LIN {X 0,Y 350.473,Z 637.276,A -85,B 0,C 180,E1 -13786.754,E2 -13786.754} C_VEL
LIN {X 0,Y 351.298,Z 630.032,A -85,B 0,C 180,E1 -13787.613,E2 -13787.613} C_VEL
LIN {X 0,Y 351.494,Z 617.509,A -85,B 0,C 180,E1 -13788.907,E2 -13788.907} C_VEL
LIN {X 0,Y 351.425,Z 604.758,A -85,B 0,C 180,E1 -13789.96,E2 -13789.96} C_VEL
LIN {X 0,Y 350.462,Z 591.602,A -85,B 0,C 180,E1 -13790.852,E2 -13790.852} C_VEL
LIN {X 0,Y 348.459,Z 578.111,A -85,B 0,C 180,E1 -13791.619,E2 -13791.619} C_VEL
LIN {X 0,Y 347.444,Z 572.402,A -85,B 0,C 180,E1 -13791.906,E2 -13791.906} C_VEL
LIN {X 0,Y 348.181,Z 560.578,A -85,B 0,C 180,E1 -13795.72,E2 -13795.72} C_VEL
LIN {X 0,Y 349.049,Z 549.243,A -85,B 0,C 180,E1 -13799.49,E2 -13799.49} C_VEL
LIN {X 0,Y 350.264,Z 537.694,A -85,B 0,C 180,E1 -13803.49,E2 -13803.49} C_VEL
LIN {X 0,Y 351.508,Z 528.335,A -85,B 0,C 180,E1 -13806.893,E2 -13806.893} C_VEL
LIN {X 0,Y 351.566,Z 524.747,A -85,B 0,C 180,E1 -13808.295,E2 -13808.295} C_VEL
LIN {X 0,Y 350.338,Z 517.421,A -85,B 0,C 180,E1 -13811.453,E2 -13811.453} C_VEL
LIN {X 0,Y 348.766,Z 509.758,A -85,B 0,C 180,E1 -13815.147,E2 -13815.147} C_VEL
LIN {X 0,Y 347.773,Z 505.172,A -85,B 0,C 180,E1 -13817.686,E2 -13817.686} C_VEL
LIN {X 0,Y 347.754,Z 505.168,A -85,B 0,C 180,E1 -13821.208,E2 -13821.208} C_VEL
LIN {X 0,Y 347.79,Z 505.161,A -85,B 0,C 180,E1 -13824.125,E2 -13824.125} C_VEL
LIN {X 0,Y 347.741,Z 505.165,A -85,B 0,C 180,E1 -13828.086,E2 -13828.086} C_VEL
LIN {X 0,Y 347.807,Z 505.155,A -85,B 0,C 180,E1 -13830.99,E2 -13830.99} C_VEL
LIN {X 0,Y 347.834,Z 505.151,A -85,B 0,C 180,E1 -13833.608,E2 -13833.608} C_VEL
LIN {X 0,Y 347.791,Z 505.156,A -85,B 0,C 180,E1 -13836.162,E2 -13836.162} C_VEL
LIN {X 0,Y 347.816,Z 505.157,A -85,B 0,C 180,E1 -13839.91,E2 -13839.91} C_VEL
LIN {X 0,Y 347.869,Z 505.148,A -85,B 0,C 180,E1 -13842.36,E2 -13842.36} C_VEL
LIN {X 0,Y 347.901,Z 505.146,A -85,B 0,C 180,E1 -13845.971,E2 -13845.971} C_VEL
LIN {X 0,Y 347.932,Z 505.144,A -85,B 0,C 180,E1 -13849.526,E2 -13849.526} C_VEL
LIN {X 0,Y 348.078,Z 505.121,A -85,B 0,C 180,E1 -13851.875,E2 -13851.875} C_VEL
LIN {X 0,Y 348.07,Z 505.128,A -85,B 0,C 180,E1 -13854.206,E2 -13854.206} C_VEL
LIN {X 0,Y 348.199,Z 505.111,A -85,B 0,C 180,E1 -13857.687,E2 -13857.687} C_VEL
LIN {X 0,Y 348.327,Z 505.096,A -85,B 0,C 180,E1 -13860,E2 -13860} C_VEL
LIN {X 0,Y 348.21,Z 505.112,A -85,B 0,C 180,E1 -13862.314,E2 -13862.314} C_VEL
LIN {X 0,Y 348.06,Z 505.128,A -85,B 0,C 180,E1 -13866.959,E2 -13866.959} C_VEL
LIN {X 0,Y 347.933,Z 505.147,A -85,B 0,C 180,E1 -13870.475,E2 -13870.475} C_VEL
LIN {X 0,Y 347.908,Z 505.299,A -85,B 0,C 180,E1 -13873.025,E2 -13873.025} C_VEL
LIN {X 0,Y 352.548,Z 517.229,A -85,B 0,C 180,E1 -13874.284,E2 -13874.284} C_VEL
LIN {X 0,Y 355.753,Z 527.322,A -85,B 0,C 180,E1 -13875.494,E2 -13875.494} C_VEL
LIN {X 0,Y 356.4,Z 530.523,A -85,B 0,C 180,E1 -13875.886,E2 -13875.886} C_VEL
LIN {X 0,Y 355.309,Z 541.181,A -85,B 0,C 180,E1 -13877.112,E2 -13877.112} C_VEL
LIN {X 0,Y 354.096,Z 551.038,A -85,B 0,C 180,E1 -13878.516,E2 -13878.516} C_VEL
LIN {X 0,Y 352.87,Z 560.144,A -85,B 0,C 180,E1 -13880.128,E2 -13880.128} C_VEL
LIN {X 0,Y 351.603,Z 568.536,A -85,B 0,C 180,E1 -13882.011,E2 -13882.011} C_VEL
LIN {X 0,Y 350.683,Z 574.262,A -85,B 0,C 180,E1 -13883.63,E2 -13883.63} C_VEL
LIN {X 0,Y 349.693,Z 579.975,A -85,B 0,C 180,E1 -13885.719,E2 -13885.719} C_VEL
LIN {X 0,Y 349.054,Z 583.768,A -85,B 0,C 180,E1 -13887.635,E2 -13887.635} C_VEL
LIN {X 0,Y 348.427,Z 586.691,A -85,B 0,C 180,E1 -13889.848,E2 -13889.848} C_VEL
LIN {X 0,Y 348.051,Z 588.043,A -85,B 0,C 180,E1 -13891.996,E2 -13891.996} C_VEL
LIN {X 0,Y 347.856,Z 588.072,A -85,B 0,C 180,E1 -13894.069,E2 -13894.069} C_VEL
LIN {X 0,Y 347.85,Z 586.893,A -85,B 0,C 180,E1 -13896.082,E2 -13896.082} C_VEL
LIN {X 0,Y 347.969,Z 584.604,A -85,B 0,C 180,E1 -13898.029,E2 -13898.029} C_VEL
LIN {X 0,Y 348.359,Z 580.571,A -85,B 0,C 180,E1 -13900.21,E2 -13900.21} C_VEL
LIN {X 0,Y 348.759,Z 576.638,A -85,B 0,C 180,E1 -13901.788,E2 -13901.788} C_VEL
LIN {X 0,Y 349.335,Z 570.93,A -85,B 0,C 180,E1 -13903.592,E2 -13903.592} C_VEL
LIN {X 0,Y 350.029,Z 563.955,A -85,B 0,C 180,E1 -13905.352,E2 -13905.352} C_VEL
LIN {X 0,Y 350.917,Z 555.421,A -85,B 0,C 180,E1 -13907.083,E2 -13907.083} C_VEL
LIN {X 0,Y 351.69,Z 546.78,A -85,B 0,C 180,E1 -13908.507,E2 -13908.507} C_VEL
LIN {X 0,Y 352.597,Z 536.445,A -85,B 0,C 180,E1 -13909.899,E2 -13909.899} C_VEL
LIN {X 0,Y 353.429,Z 525.889,A -85,B 0,C 180,E1 -13911.051,E2 -13911.051} C_VEL
LIN {X 0,Y 351.915,Z 519.372,A -85,B 0,C 180,E1 -13911.75,E2 -13911.75} C_VEL
LIN {X 0,Y 348.274,Z 506.984,A -85,B 0,C 180,E1 -13912.914,E2 -13912.914} C_VEL
LIN {X 0,Y 347.785,Z 505.165,A -85,B 0,C 180,E1 -13913.066,E2 -13913.066} C_VEL
LIN {X 0,Y 347.738,Z 505.168,A -85,B 0,C 180,E1 -13916.928,E2 -13916.928} C_VEL
LIN {X 0,Y 347.81,Z 505.16,A -85,B 0,C 180,E1 -13920.99,E2 -13920.99} C_VEL
LIN {X 0,Y 347.836,Z 505.158,A -85,B 0,C 180,E1 -13923.608,E2 -13923.608} C_VEL
LIN {X 0,Y 347.79,Z 505.16,A -85,B 0,C 180,E1 -13926.162,E2 -13926.162} C_VEL
LIN {X 0,Y 347.805,Z 505.16,A -85,B 0,C 180,E1 -13929.909,E2 -13929.909} C_VEL
LIN {X 0,Y 347.837,Z 505.158,A -85,B 0,C 180,E1 -13933.568,E2 -13933.568} C_VEL
LIN {X 0,Y 347.895,Z 505.151,A -85,B 0,C 180,E1 -13937.161,E2 -13937.161} C_VEL
LIN {X 0,Y 347.94,Z 505.142,A -85,B 0,C 180,E1 -13940.701,E2 -13940.701} C_VEL
LIN {X 0,Y 348.049,Z 505.128,A -85,B 0,C 180,E1 -13944.205,E2 -13944.205} C_VEL
LIN {X 0,Y 348.211,Z 505.11,A -85,B 0,C 180,E1 -13947.686,E2 -13947.686} C_VEL
LIN {X 0,Y 348.268,Z 505.101,A -85,B 0,C 180,E1 -13950,E2 -13950} C_VEL
LIN {X 0,Y 348.208,Z 505.108,A -85,B 0,C 180,E1 -13952.313,E2 -13952.313} C_VEL
LIN {X 0,Y 348.061,Z 505.129,A -85,B 0,C 180,E1 -13956.958,E2 -13956.958} C_VEL
LIN {X 0,Y 347.901,Z 505.147,A -85,B 0,C 180,E1 -13960.475,E2 -13960.475} C_VEL
LIN {X 0,Y 347.903,Z 505.146,A -85,B 0,C 180,E1 -13964.15,E2 -13964.15} C_VEL
LIN {X 0,Y 347.834,Z 505.155,A -85,B 0,C 180,E1 -13968.259,E2 -13968.259} C_VEL
LIN {X 0,Y 347.792,Z 505.162,A -85,B 0,C 180,E1 -13971.634,E2 -13971.634} C_VEL
LIN {X 0,Y 347.798,Z 505.164,A -85,B 0,C 180,E1 -13975.11,E2 -13975.11} C_VEL
LIN {X 0,Y 347.761,Z 505.168,A -85,B 0,C 180,E1 -13979.014,E2 -13979.014} C_VEL
LIN {X 0,Y 347.737,Z 505.172,A -85,B 0,C 180,E1 -13983.072,E2 -13983.072} C_VEL
LIN {X 0,Y 347.773,Z 505.162,A -85,B 0,C 180,E1 -13986.065,E2 -13986.065} C_VEL
LIN {X 0,Y 347.734,Z 505.17,A -85,B 0,C 180,E1 -13988.795,E2 -13988.795} C_VEL
LIN {X 0,Y 347.746,Z 505.166,A -85,B 0,C 180,E1 -13991.831,E2 -13991.831} C_VEL
LIN {X 0,Y 347.708,Z 505.176,A -85,B 0,C 180,E1 -13995.026,E2 -13995.026} C_VEL
LIN {X 0,Y 347.752,Z 505.165,A -85,B 0,C 180,E1 -13998.397,E2 -13998.397} C_VEL
LIN {X 0,Y 347.775,Z 505.162,A -85,B 0,C 180,E1 -14002.011,E2 -14002.011} C_VEL
LIN {X 0,Y 347.752,Z 505.165,A -85,B 0,C 180,E1 -14002.91,E2 -14002.91} C_VEL
LIN {X 0,Y 347.07,Z 505.25,A -85,B 0,C 180,E1 -14003.877,E2 -14003.877} C_VEL
LIN {X 0,Y 344.218,Z 505.607,A -85,B 0,C 180,E1 -14005.45,E2 -14005.45} C_VEL
LIN {X 0,Y 341.807,Z 505.908,A -85,B 0,C 180,E1 -14006.724,E2 -14006.724} C_VEL
LIN {X 0,Y 340.769,Z 506.036,A -85,B 0,C 180,E1 -14007.709,E2 -14007.709} C_VEL
LIN {X 0,Y 340.682,Z 506.045,A -85,B 0,C 180,E1 -14008.042,E2 -14008.042} C_VEL
LIN {X 0,Y 340.777,Z 506.034,A -85,B 0,C 180,E1 -14010.332,E2 -14010.332} C_VEL
LIN {X 0,Y 340.806,Z 506.035,A -85,B 0,C 180,E1 -14013.02,E2 -14013.02} C_VEL
LIN {X 0,Y 340.757,Z 506.037,A -85,B 0,C 180,E1 -14015.638,E2 -14015.638} C_VEL
LIN {X 0,Y 340.737,Z 506.04,A -85,B 0,C 180,E1 -14019.473,E2 -14019.473} C_VEL
LIN {X 0,Y 340.86,Z 506.023,A -85,B 0,C 180,E1 -14021.984,E2 -14021.984} C_VEL
LIN {X 0,Y 340.872,Z 506.022,A -85,B 0,C 180,E1 -14025.705,E2 -14025.705} C_VEL
LIN {X 0,Y 340.851,Z 506.027,A -85,B 0,C 180,E1 -14029.305,E2 -14029.305} C_VEL
LIN {X 0,Y 341.018,Z 506.009,A -85,B 0,C 180,E1 -14032.897,E2 -14032.897} C_VEL
LIN {X 0,Y 341.167,Z 505.985,A -85,B 0,C 180,E1 -14037.638,E2 -14037.638} C_VEL
LIN {X 0,Y 341.256,Z 505.974,A -85,B 0,C 180,E1 -14040,E2 -14040} C_VEL
LIN {X 0,Y 341.157,Z 505.987,A -85,B 0,C 180,E1 -14042.361,E2 -14042.361} C_VEL
LIN {X 0,Y 341.005,Z 506.009,A -85,B 0,C 180,E1 -14047.103,E2 -14047.103} C_VEL
LIN {X 0,Y 340.875,Z 506.026,A -85,B 0,C 180,E1 -14050.693,E2 -14050.693} C_VEL
LIN {X 0,Y 340.864,Z 506.024,A -85,B 0,C 180,E1 -14054.325,E2 -14054.325} C_VEL
LIN {X 0,Y 340.787,Z 506.035,A -85,B 0,C 180,E1 -14058.44,E2 -14058.44} C_VEL
LIN {X 0,Y 340.718,Z 506.041,A -85,B 0,C 180,E1 -14061.841,E2 -14061.841} C_VEL
LIN {X 0,Y 340.753,Z 506.042,A -85,B 0,C 180,E1 -14064.838,E2 -14064.838} C_VEL
LIN {X 0,Y 340.685,Z 506.047,A -85,B 0,C 180,E1 -14068.324,E2 -14068.324} C_VEL
LIN {X 0,Y 340.695,Z 506.047,A -85,B 0,C 180,E1 -14071.045,E2 -14071.045} C_VEL
LIN {X 0,Y 340.719,Z 506.042,A -85,B 0,C 180,E1 -14075.279,E2 -14075.279} C_VEL
LIN {X 0,Y 340.71,Z 506.044,A -85,B 0,C 180,E1 -14078.386,E2 -14078.386} C_VEL
LIN {X 0,Y 340.722,Z 506.044,A -85,B 0,C 180,E1 -14082.05,E2 -14082.05} C_VEL
LIN {X 0,Y 340.732,Z 506.146,A -85,B 0,C 180,E1 -14083.083,E2 -14083.083} C_VEL
LIN {X 0,Y 342.406,Z 514.631,A -85,B 0,C 180,E1 -14086.698,E2 -14086.698} C_VEL
LIN {X 0,Y 344.43,Z 524.949,A -85,B 0,C 180,E1 -14090.839,E2 -14090.839} C_VEL
LIN {X 0,Y 344.982,Z 528.832,A -85,B 0,C 180,E1 -14092.326,E2 -14092.326} C_VEL
LIN {X 0,Y 343.768,Z 538.566,A -85,B 0,C 180,E1 -14095.791,E2 -14095.791} C_VEL
LIN {X 0,Y 342.707,Z 548.225,A -85,B 0,C 180,E1 -14099.157,E2 -14099.157} C_VEL
LIN {X 0,Y 341.579,Z 559.744,A -85,B 0,C 180,E1 -14103.086,E2 -14103.086} C_VEL
LIN {X 0,Y 340.865,Z 569.197,A -85,B 0,C 180,E1 -14106.293,E2 -14106.293} C_VEL
LIN {X 0,Y 340.337,Z 578.292,A -85,B 0,C 180,E1 -14109.33,E2 -14109.33} C_VEL
LIN {X 0,Y 341.93,Z 594.59,A -85,B 0,C 180,E1 -14110.059,E2 -14110.059} C_VEL
LIN {X 0,Y 342.857,Z 607.272,A -85,B 0,C 180,E1 -14110.854,E2 -14110.854} C_VEL
LIN {X 0,Y 343.382,Z 619.211,A -85,B 0,C 180,E1 -14111.813,E2 -14111.813} C_VEL
LIN {X 0,Y 343.553,Z 630.124,A -85,B 0,C 180,E1 -14112.898,E2 -14112.898} C_VEL
LIN {X 0,Y 342.443,Z 641.064,A -85,B 0,C 180,E1 -14114.221,E2 -14114.221} C_VEL
LIN {X 0,Y 341.276,Z 650.865,A -85,B 0,C 180,E1 -14115.693,E2 -14115.693} C_VEL
LIN {X 0,Y 340.669,Z 659,A -85,B 0,C 180,E1 -14117.187,E2 -14117.187} C_VEL
LIN {X 0,Y 340.11,Z 666.98,A -85,B 0,C 180,E1 -14118.981,E2 -14118.981} C_VEL
LIN {X 0,Y 339.896,Z 672.392,A -85,B 0,C 180,E1 -14120.479,E2 -14120.479} C_VEL
LIN {X 0,Y 339.828,Z 677.665,A -85,B 0,C 180,E1 -14122.275,E2 -14122.275} C_VEL
LIN {X 0,Y 339.909,Z 681.718,A -85,B 0,C 180,E1 -14124.066,E2 -14124.066} C_VEL
LIN {X 0,Y 340.118,Z 683.798,A -85,B 0,C 180,E1 -14125.259,E2 -14125.259} C_VEL
LIN {X 0,Y 340.201,Z 685.4,A -85,B 0,C 180,E1 -14126.447,E2 -14126.447} C_VEL
LIN {X 0,Y 340.266,Z 686.567,A -85,B 0,C 180,E1 -14127.633,E2 -14127.633} C_VEL
LIN {X 0,Y 340.349,Z 687.288,A -85,B 0,C 180,E1 -14128.817,E2 -14128.817} C_VEL
LIN {X 0,Y 340.592,Z 687.577,A -85,B 0,C 180,E1 -14130,E2 -14130} C_VEL
LIN {X 0,Y 340.228,Z 686.787,A -85,B 0,C 180,E1 -14132.368,E2 -14132.368} C_VEL
LIN {X 0,Y 340.156,Z 685.761,A -85,B 0,C 180,E1 -14133.554,E2 -14133.554} C_VEL
LIN {X 0,Y 340.047,Z 684.276,A -85,B 0,C 180,E1 -14134.742,E2 -14134.742} C_VEL
LIN {X 0,Y 339.813,Z 680.445,A -85,B 0,C 180,E1 -14136.911,E2 -14136.911} C_VEL
LIN {X 0,Y 339.76,Z 675.519,A -85,B 0,C 180,E1 -14138.925,E2 -14138.925} C_VEL
LIN {X 0,Y 340.024,Z 668.793,A -85,B 0,C 180,E1 -14141.022,E2 -14141.022} C_VEL
LIN {X 0,Y 340.615,Z 661.62,A -85,B 0,C 180,E1 -14142.815,E2 -14142.815} C_VEL
LIN {X 0,Y 341.278,Z 654.418,A -85,B 0,C 180,E1 -14144.307,E2 -14144.307} C_VEL
LIN {X 0,Y 342.446,Z 645.887,A -85,B 0,C 180,E1 -14145.779,E2 -14145.779} C_VEL
LIN {X 0,Y 343.801,Z 635.622,A -85,B 0,C 180,E1 -14147.242,E2 -14147.242} C_VEL
LIN {X 0,Y 344.405,Z 629.581,A -85,B 0,C 180,E1 -14147.978,E2 -14147.978} C_VEL
LIN {X 0,Y 344.686,Z 617.338,A -85,B 0,C 180,E1 -14149.283,E2 -14149.283} C_VEL
LIN {X 0,Y 344.676,Z 604.209,A -85,B 0,C 180,E1 -14150.421,E2 -14150.421} C_VEL
LIN {X 0,Y 343.701,Z 591.118,A -85,B 0,C 180,E1 -14151.354,E2 -14151.354} C_VEL
LIN {X 0,Y 341.775,Z 578.056,A -85,B 0,C 180,E1 -14152.133,E2 -14152.133} C_VEL
LIN {X 0,Y 340.468,Z 571.091,A -85,B 0,C 180,E1 -14152.513,E2 -14152.513} C_VEL
LIN {X 0,Y 341.243,Z 559.73,A -85,B 0,C 180,E1 -14156.283,E2 -14156.283} C_VEL
LIN {X 0,Y 342.145,Z 548.945,A -85,B 0,C 180,E1 -14159.978,E2 -14159.978} C_VEL
LIN {X 0,Y 343.488,Z 537.019,A -85,B 0,C 180,E1 -14164.241,E2 -14164.241} C_VEL
LIN {X 0,Y 344.649,Z 528.824,A -85,B 0,C 180,E1 -14167.319,E2 -14167.319} C_VEL
LIN {X 0,Y 344.36,Z 524.396,A -85,B 0,C 180,E1 -14169.146,E2 -14169.146} C_VEL
LIN {X 0,Y 343.367,Z 518.76,A -85,B 0,C 180,E1 -14171.676,E2 -14171.676} C_VEL
LIN {X 0,Y 342.021,Z 512.107,A -85,B 0,C 180,E1 -14174.958,E2 -14174.958} C_VEL
LIN {X 0,Y 340.716,Z 506.047,A -85,B 0,C 180,E1 -14178.401,E2 -14178.401} C_VEL
LIN {X 0,Y 340.735,Z 506.04,A -85,B 0,C 180,E1 -14181.773,E2 -14181.773} C_VEL
LIN {X 0,Y 340.725,Z 506.04,A -85,B 0,C 180,E1 -14185.596,E2 -14185.596} C_VEL
LIN {X 0,Y 340.706,Z 506.044,A -85,B 0,C 180,E1 -14188.956,E2 -14188.956} C_VEL
LIN {X 0,Y 340.781,Z 506.033,A -85,B 0,C 180,E1 -14192.474,E2 -14192.474} C_VEL
LIN {X 0,Y 340.759,Z 506.034,A -85,B 0,C 180,E1 -14195.639,E2 -14195.639} C_VEL
LIN {X 0,Y 340.748,Z 506.035,A -85,B 0,C 180,E1 -14199.474,E2 -14199.474} C_VEL
LIN {X 0,Y 340.861,Z 506.021,A -85,B 0,C 180,E1 -14201.985,E2 -14201.985} C_VEL
LIN {X 0,Y 340.872,Z 506.019,A -85,B 0,C 180,E1 -14205.705,E2 -14205.705} C_VEL
LIN {X 0,Y 340.874,Z 506.022,A -85,B 0,C 180,E1 -14209.307,E2 -14209.307} C_VEL
LIN {X 0,Y 341.08,Z 505.998,A -85,B 0,C 180,E1 -14212.899,E2 -14212.899} C_VEL
LIN {X 0,Y 341.16,Z 505.988,A -85,B 0,C 180,E1 -14217.639,E2 -14217.639} C_VEL
LIN {X 0,Y 341.278,Z 505.974,A -85,B 0,C 180,E1 -14220,E2 -14220} C_VEL
LIN {X 0,Y 341.171,Z 505.989,A -85,B 0,C 180,E1 -14222.362,E2 -14222.362} C_VEL
LIN {X 0,Y 341.007,Z 506.008,A -85,B 0,C 180,E1 -14227.104,E2 -14227.104} C_VEL
LIN {X 0,Y 340.875,Z 506.024,A -85,B 0,C 180,E1 -14230.694,E2 -14230.694} C_VEL
LIN {X 0,Y 340.834,Z 506.032,A -85,B 0,C 180,E1 -14232.391,E2 -14232.391} C_VEL
LIN {X 0,Y 345.864,Z 518.784,A -85,B 0,C 180,E1 -14233.814,E2 -14233.814} C_VEL
LIN {X 0,Y 349.288,Z 529.538,A -85,B 0,C 180,E1 -14235.164,E2 -14235.164} C_VEL
LIN {X 0,Y 349.813,Z 531.661,A -85,B 0,C 180,E1 -14235.439,E2 -14235.439} C_VEL
LIN {X 0,Y 348.79,Z 542.242,A -85,B 0,C 180,E1 -14236.687,E2 -14236.687} C_VEL
LIN {X 0,Y 347.519,Z 552.016,A -85,B 0,C 180,E1 -14238.102,E2 -14238.102} C_VEL
LIN {X 0,Y 346.371,Z 560.192,A -85,B 0,C 180,E1 -14239.56,E2 -14239.56} C_VEL
LIN {X 0,Y 345.16,Z 567.907,A -85,B 0,C 180,E1 -14241.256,E2 -14241.256} C_VEL
LIN {X 0,Y 343.974,Z 574.75,A -85,B 0,C 180,E1 -14243.156,E2 -14243.156} C_VEL
LIN {X 0,Y 343.15,Z 579.49,A -85,B 0,C 180,E1 -14244.826,E2 -14244.826} C_VEL
LIN {X 0,Y 342.324,Z 583.875,A -85,B 0,C 180,E1 -14246.851,E2 -14246.851} C_VEL
LIN {X 0,Y 341.878,Z 586.041,A -85,B 0,C 180,E1 -14248.218,E2 -14248.218} C_VEL
LIN {X 0,Y 341.361,Z 588.143,A -85,B 0,C 180,E1 -14250.15,E2 -14250.15} C_VEL
LIN {X 0,Y 340.993,Z 589.24,A -85,B 0,C 180,E1 -14252.404,E2 -14252.404} C_VEL
LIN {X 0,Y 340.821,Z 588.999,A -85,B 0,C 180,E1 -14254.428,E2 -14254.428} C_VEL
LIN {X 0,Y 340.852,Z 587.273,A -85,B 0,C 180,E1 -14256.724,E2 -14256.724} C_VEL
LIN {X 0,Y 341.075,Z 584.079,A -85,B 0,C 180,E1 -14259.009,E2 -14259.009} C_VEL
LIN {X 0,Y 341.594,Z 579.461,A -85,B 0,C 180,E1 -14261.177,E2 -14261.177} C_VEL
LIN {X 0,Y 342.121,Z 574.168,A -85,B 0,C 180,E1 -14263.046,E2 -14263.046} C_VEL
LIN {X 0,Y 342.807,Z 567.072,A -85,B 0,C 180,E1 -14265.016,E2 -14265.016} C_VEL
LIN {X 0,Y 343.716,Z 559.11,A -85,B 0,C 180,E1 -14266.755,E2 -14266.755} C_VEL
LIN {X 0,Y 344.631,Z 549.858,A -85,B 0,C 180,E1 -14268.4,E2 -14268.4} C_VEL
LIN {X 0,Y 345.554,Z 539.634,A -85,B 0,C 180,E1 -14269.871,E2 -14269.871} C_VEL
LIN {X 0,Y 346.414,Z 528.922,A -85,B 0,C 180,E1 -14271.11,E2 -14271.11} C_VEL
LIN {X 0,Y 346.459,Z 526.116,A -85,B 0,C 180,E1 -14271.408,E2 -14271.408} C_VEL
LIN {X 0,Y 343.188,Z 514.342,A -85,B 0,C 180,E1 -14272.65,E2 -14272.65} C_VEL
LIN {X 0,Y 340.757,Z 506.041,A -85,B 0,C 180,E1 -14273.413,E2 -14273.413} C_VEL
LIN {X 0,Y 340.697,Z 506.044,A -85,B 0,C 180,E1 -14276.153,E2 -14276.153} C_VEL
LIN {X 0,Y 340.779,Z 506.033,A -85,B 0,C 180,E1 -14280.333,E2 -14280.333} C_VEL
LIN {X 0,Y 340.809,Z 506.032,A -85,B 0,C 180,E1 -14283.02,E2 -14283.02} C_VEL
LIN {X 0,Y 340.759,Z 506.039,A -85,B 0,C 180,E1 -14285.638,E2 -14285.638} C_VEL
LIN {X 0,Y 340.735,Z 506.044,A -85,B 0,C 180,E1 -14289.473,E2 -14289.473} C_VEL
LIN {X 0,Y 340.797,Z 506.032,A -85,B 0,C 180,E1 -14291.981,E2 -14291.981} C_VEL
LIN {X 0,Y 340.874,Z 506.024,A -85,B 0,C 180,E1 -14295.705,E2 -14295.705} C_VEL
LIN {X 0,Y 340.854,Z 506.029,A -85,B 0,C 180,E1 -14299.305,E2 -14299.305} C_VEL
LIN {X 0,Y 341.008,Z 506.007,A -85,B 0,C 180,E1 -14302.897,E2 -14302.897} C_VEL
LIN {X 0,Y 341.172,Z 505.987,A -85,B 0,C 180,E1 -14307.639,E2 -14307.639} C_VEL
LIN {X 0,Y 341.221,Z 505.979,A -85,B 0,C 180,E1 -14310,E2 -14310} C_VEL
LIN {X 0,Y 341.169,Z 505.985,A -85,B 0,C 180,E1 -14312.361,E2 -14312.361} C_VEL
LIN {X 0,Y 341.008,Z 506.009,A -85,B 0,C 180,E1 -14317.103,E2 -14317.103} C_VEL
LIN {X 0,Y 340.853,Z 506.025,A -85,B 0,C 180,E1 -14320.694,E2 -14320.694} C_VEL
LIN {X 0,Y 340.868,Z 506.022,A -85,B 0,C 180,E1 -14324.325,E2 -14324.325} C_VEL
LIN {X 0,Y 340.791,Z 506.032,A -85,B 0,C 180,E1 -14328.44,E2 -14328.44} C_VEL
LIN {X 0,Y 340.758,Z 506.037,A -85,B 0,C 180,E1 -14331.857,E2 -14331.857} C_VEL
LIN {X 0,Y 340.749,Z 506.038,A -85,B 0,C 180,E1 -14335.666,E2 -14335.666} C_VEL
LIN {X 0,Y 340.735,Z 506.04,A -85,B 0,C 180,E1 -14339.671,E2 -14339.671} C_VEL
LIN {X 0,Y 340.696,Z 506.044,A -85,B 0,C 180,E1 -14343.846,E2 -14343.846} C_VEL
LIN {X 0,Y 340.706,Z 506.045,A -85,B 0,C 180,E1 -14346.742,E2 -14346.742} C_VEL
LIN {X 0,Y 340.654,Z 506.049,A -85,B 0,C 180,E1 -14350.239,E2 -14350.239} C_VEL
LIN {X 0,Y 340.676,Z 506.05,A -85,B 0,C 180,E1 -14352.904,E2 -14352.904} C_VEL
LIN {X 0,Y 340.678,Z 506.051,A -85,B 0,C 180,E1 -14357.095,E2 -14357.095} C_VEL
LIN {X 0,Y 340.701,Z 506.043,A -85,B 0,C 180,E1 -14360.247,E2 -14360.247} C_VEL
LIN {X 0,Y 340.712,Z 506.043,A -85,B 0,C 180,E1 -14363.559,E2 -14363.559} C_VEL
LIN {X 0,Y 340.695,Z 506.044,A -85,B 0,C 180,E1 -14366.153,E2 -14366.153} C_VEL
LIN {X 0,Y 340.682,Z 506.045,A -85,B 0,C 180,E1 -14368.042,E2 -14368.042} C_VEL
LIN {X 0,Y 340.013,Z 506.134,A -85,B 0,C 180,E1 -14369.029,E2 -14369.029} C_VEL
LIN {X 0,Y 337.185,Z 506.483,A -85,B 0,C 180,E1 -14370.636,E2 -14370.636} C_VEL
LIN {X 0,Y 334.803,Z 506.777,A -85,B 0,C 180,E1 -14371.937,E2 -14371.937} C_VEL
LIN {X 0,Y 333.794,Z 506.908,A -85,B 0,C 180,E1 -14372.943,E2 -14372.943} C_VEL
LIN {X 0,Y 333.719,Z 506.91,A -85,B 0,C 180,E1 -14373.284,E2 -14373.284} C_VEL
LIN {X 0,Y 333.671,Z 506.919,A -85,B 0,C 180,E1 -14376.409,E2 -14376.409} C_VEL
LIN {X 0,Y 333.734,Z 506.911,A -85,B 0,C 180,E1 -14380.309,E2 -14380.309} C_VEL
LIN {X 0,Y 333.75,Z 506.913,A -85,B 0,C 180,E1 -14382.854,E2 -14382.854} C_VEL
LIN {X 0,Y 333.799,Z 506.905,A -85,B 0,C 180,E1 -14386.608,E2 -14386.608} C_VEL
LIN {X 0,Y 333.822,Z 506.9,A -85,B 0,C 180,E1 -14390.303,E2 -14390.303} C_VEL
LIN {X 0,Y 334,Z 506.877,A -85,B 0,C 180,E1 -14393.96,E2 -14393.96} C_VEL
LIN {X 0,Y 334.104,Z 506.865,A -85,B 0,C 180,E1 -14397.588,E2 -14397.588} C_VEL
LIN {X 0,Y 334.208,Z 506.852,A -85,B 0,C 180,E1 -14400,E2 -14400} C_VEL
LIN {X 0,Y 334.094,Z 506.867,A -85,B 0,C 180,E1 -14402.411,E2 -14402.411} C_VEL
LIN {X 0,Y 333.992,Z 506.879,A -85,B 0,C 180,E1 -14406.039,E2 -14406.039} C_VEL
LIN {X 0,Y 333.852,Z 506.896,A -85,B 0,C 180,E1 -14409.695,E2 -14409.695} C_VEL
LIN {X 0,Y 333.8,Z 506.904,A -85,B 0,C 180,E1 -14413.391,E2 -14413.391} C_VEL
LIN {X 0,Y 333.721,Z 506.915,A -85,B 0,C 180,E1 -14417.147,E2 -14417.147} C_VEL
LIN {X 0,Y 333.686,Z 506.916,A -85,B 0,C 180,E1 -14419.693,E2 -14419.693} C_VEL
LIN {X 0,Y 333.669,Z 506.919,A -85,B 0,C 180,E1 -14423.59,E2 -14423.59} C_VEL
LIN {X 0,Y 333.663,Z 506.921,A -85,B 0,C 180,E1 -14426.252,E2 -14426.252} C_VEL
LIN {X 0,Y 333.662,Z 506.921,A -85,B 0,C 180,E1 -14430.277,E2 -14430.277} C_VEL
LIN {X 0,Y 333.637,Z 506.925,A -85,B 0,C 180,E1 -14433.208,E2 -14433.208} C_VEL
LIN {X 0,Y 333.676,Z 506.919,A -85,B 0,C 180,E1 -14436.139,E2 -14436.139} C_VEL
LIN {X 0,Y 333.647,Z 506.926,A -85,B 0,C 180,E1 -14439.192,E2 -14439.192} C_VEL
LIN {X 0,Y 333.694,Z 506.983,A -85,B 0,C 180,E1 -14442.707,E2 -14442.707} C_VEL
LIN {X 0,Y 335.435,Z 515.963,A -85,B 0,C 180,E1 -14446.603,E2 -14446.603} C_VEL
LIN {X 0,Y 337.265,Z 525.299,A -85,B 0,C 180,E1 -14450.445,E2 -14450.445} C_VEL
LIN {X 0,Y 337.961,Z 529.782,A -85,B 0,C 180,E1 -14452.206,E2 -14452.206} C_VEL
LIN {X 0,Y 337.023,Z 537.529,A -85,B 0,C 180,E1 -14455.033,E2 -14455.033} C_VEL
LIN {X 0,Y 335.881,Z 547.115,A -85,B 0,C 180,E1 -14458.459,E2 -14458.459} C_VEL
LIN {X 0,Y 334.487,Z 560.458,A -85,B 0,C 180,E1 -14463.145,E2 -14463.145} C_VEL
LIN {X 0,Y 333.725,Z 569.923,A -85,B 0,C 180,E1 -14466.414,E2 -14466.414} C_VEL
LIN {X 0,Y 333.3,Z 577.675,A -85,B 0,C 180,E1 -14468.994,E2 -14468.994} C_VEL
LIN {X 0,Y 334.772,Z 592.359,A -85,B 0,C 180,E1 -14469.643,E2 -14469.643} C_VEL
LIN {X 0,Y 335.779,Z 605.034,A -85,B 0,C 180,E1 -14470.434,E2 -14470.434} C_VEL
LIN {X 0,Y 336.351,Z 617.38,A -85,B 0,C 180,E1 -14471.432,E2 -14471.432} C_VEL
LIN {X 0,Y 336.552,Z 629.762,A -85,B 0,C 180,E1 -14472.688,E2 -14472.688} C_VEL
LIN {X 0,Y 335.413,Z 640.55,A -85,B 0,C 180,E1 -14474.037,E2 -14474.037} C_VEL
LIN {X 0,Y 334.402,Z 649.393,A -85,B 0,C 180,E1 -14475.392,E2 -14475.392} C_VEL
LIN {X 0,Y 333.686,Z 657.589,A -85,B 0,C 180,E1 -14476.914,E2 -14476.914} C_VEL
LIN {X 0,Y 333.099,Z 665.646,A -85,B 0,C 180,E1 -14478.746,E2 -14478.746} C_VEL
LIN {X 0,Y 332.854,Z 671.104,A -85,B 0,C 180,E1 -14480.275,E2 -14480.275} C_VEL
LIN {X 0,Y 332.765,Z 676.431,A -85,B 0,C 180,E1 -14482.11,E2 -14482.11} C_VEL
LIN {X 0,Y 332.854,Z 680.536,A -85,B 0,C 180,E1 -14483.94,E2 -14483.94} C_VEL
LIN {X 0,Y 333.055,Z 682.656,A -85,B 0,C 180,E1 -14485.158,E2 -14485.158} C_VEL
LIN {X 0,Y 333.156,Z 684.282,A -85,B 0,C 180,E1 -14486.372,E2 -14486.372} C_VEL
LIN {X 0,Y 333.233,Z 685.467,A -85,B 0,C 180,E1 -14487.583,E2 -14487.583} C_VEL
LIN {X 0,Y 333.32,Z 686.221,A -85,B 0,C 180,E1 -14488.792,E2 -14488.792} C_VEL
LIN {X 0,Y 333.565,Z 686.531,A -85,B 0,C 180,E1 -14490,E2 -14490} C_VEL
LIN {X 0,Y 333.185,Z 685.765,A -85,B 0,C 180,E1 -14492.418,E2 -14492.418} C_VEL
LIN {X 0,Y 333.108,Z 684.768,A -85,B 0,C 180,E1 -14493.629,E2 -14493.629} C_VEL
LIN {X 0,Y 332.985,Z 683.295,A -85,B 0,C 180,E1 -14494.843,E2 -14494.843} C_VEL
LIN {X 0,Y 332.739,Z 679.768,A -85,B 0,C 180,E1 -14496.918,E2 -14496.918} C_VEL
LIN {X 0,Y 332.7,Z 674.608,A -85,B 0,C 180,E1 -14499.116,E2 -14499.116} C_VEL
LIN {X 0,Y 333.013,Z 667.97,A -85,B 0,C 180,E1 -14501.257,E2 -14501.257} C_VEL
LIN {X 0,Y 333.796,Z 659.528,A -85,B 0,C 180,E1 -14503.392,E2 -14503.392} C_VEL
LIN {X 0,Y 334.746,Z 650.846,A -85,B 0,C 180,E1 -14505.153,E2 -14505.153} C_VEL
LIN {X 0,Y 336.201,Z 640.391,A -85,B 0,C 180,E1 -14506.861,E2 -14506.861} C_VEL
LIN {X 0,Y 337.453,Z 631.602,A -85,B 0,C 180,E1 -14508.047,E2 -14508.047} C_VEL
LIN {X 0,Y 337.845,Z 619.651,A -85,B 0,C 180,E1 -14509.441,E2 -14509.441} C_VEL
LIN {X 0,Y 338.023,Z 608.428,A -85,B 0,C 180,E1 -14510.508,E2 -14510.508} C_VEL
LIN {X 0,Y 337.381,Z 594.985,A -85,B 0,C 180,E1 -14511.572,E2 -14511.572} C_VEL
LIN {X 0,Y 335.593,Z 580.952,A -85,B 0,C 180,E1 -14512.509,E2 -14512.509} C_VEL
LIN {X 0,Y 333.477,Z 569.8,A -85,B 0,C 180,E1 -14513.153,E2 -14513.153} C_VEL
LIN {X 0,Y 334.316,Z 558.919,A -85,B 0,C 180,E1 -14516.871,E2 -14516.871} C_VEL
LIN {X 0,Y 335.31,Z 547.924,A -85,B 0,C 180,E1 -14520.757,E2 -14520.757} C_VEL
LIN {X 0,Y 336.517,Z 538.218,A -85,B 0,C 180,E1 -14524.325,E2 -14524.325} C_VEL
LIN {X 0,Y 337.61,Z 530.9,A -85,B 0,C 180,E1 -14527.135,E2 -14527.135} C_VEL
LIN {X 0,Y 337.741,Z 528.449,A -85,B 0,C 180,E1 -14528.125,E2 -14528.125} C_VEL
LIN {X 0,Y 336.876,Z 522.501,A -85,B 0,C 180,E1 -14530.769,E2 -14530.769} C_VEL
LIN {X 0,Y 335.357,Z 514.811,A -85,B 0,C 180,E1 -14534.559,E2 -14534.559} C_VEL
LIN {X 0,Y 333.875,Z 507.891,A -85,B 0,C 180,E1 -14538.466,E2 -14538.466} C_VEL
LIN {X 0,Y 333.658,Z 506.928,A -85,B 0,C 180,E1 -14539.135,E2 -14539.135} C_VEL
LIN {X 0,Y 333.667,Z 506.922,A -85,B 0,C 180,E1 -14543.168,E2 -14543.168} C_VEL
LIN {X 0,Y 333.676,Z 506.92,A -85,B 0,C 180,E1 -14545.342,E2 -14545.342} C_VEL
LIN {X 0,Y 333.705,Z 506.917,A -85,B 0,C 180,E1 -14549.711,E2 -14549.711} C_VEL
LIN {X 0,Y 333.746,Z 506.91,A -85,B 0,C 180,E1 -14552.402,E2 -14552.402} C_VEL
LIN {X 0,Y 333.73,Z 506.912,A -85,B 0,C 180,E1 -14555.091,E2 -14555.091} C_VEL
LIN {X 0,Y 333.683,Z 506.913,A -85,B 0,C 180,E1 -14559.02,E2 -14559.02} C_VEL
LIN {X 0,Y 333.797,Z 506.902,A -85,B 0,C 180,E1 -14561.59,E2 -14561.59} C_VEL
LIN {X 0,Y 333.811,Z 506.898,A -85,B 0,C 180,E1 -14565.577,E2 -14565.577} C_VEL
LIN {X 0,Y 333.837,Z 506.896,A -85,B 0,C 180,E1 -14569.078,E2 -14569.078} C_VEL
LIN {X 0,Y 334.03,Z 506.875,A -85,B 0,C 180,E1 -14572.748,E2 -14572.748} C_VEL
LIN {X 0,Y 333.802,Z 506.898,A -85,B 0,C 180,E1 -14575.169,E2 -14575.169} C_VEL
LIN {X 0,Y 334.097,Z 506.868,A -85,B 0,C 180,E1 -14577.589,E2 -14577.589} C_VEL
LIN {X 0,Y 334.23,Z 506.852,A -85,B 0,C 180,E1 -14580,E2 -14580} C_VEL
LIN {X 0,Y 334.108,Z 506.869,A -85,B 0,C 180,E1 -14582.411,E2 -14582.411} C_VEL
LIN {X 0,Y 333.965,Z 506.88,A -85,B 0,C 180,E1 -14586.519,E2 -14586.519} C_VEL
LIN {X 0,Y 333.853,Z 506.899,A -85,B 0,C 180,E1 -14589.696,E2 -14589.696} C_VEL
LIN {X 0,Y 333.834,Z 507.045,A -85,B 0,C 180,E1 -14591.768,E2 -14591.768} C_VEL
LIN {X 0,Y 335.565,Z 511.441,A -85,B 0,C 180,E1 -14592.243,E2 -14592.243} C_VEL
LIN {X 0,Y 339.671,Z 521.644,A -85,B 0,C 180,E1 -14593.476,E2 -14593.476} C_VEL
LIN {X 0,Y 342.88,Z 531.995,A -85,B 0,C 180,E1 -14594.846,E2 -14594.846} C_VEL
LIN {X 0,Y 343.322,Z 534.063,A -85,B 0,C 180,E1 -14595.13,E2 -14595.13} C_VEL
LIN {X 0,Y 341.99,Z 545.584,A -85,B 0,C 180,E1 -14596.552,E2 -14596.552} C_VEL
LIN {X 0,Y 340.676,Z 555.116,A -85,B 0,C 180,E1 -14598.026,E2 -14598.026} C_VEL
LIN {X 0,Y 339.337,Z 563.654,A -85,B 0,C 180,E1 -14599.667,E2 -14599.667} C_VEL
LIN {X 0,Y 338.168,Z 570.687,A -85,B 0,C 180,E1 -14601.341,E2 -14601.341} C_VEL
LIN {X 0,Y 336.934,Z 577.384,A -85,B 0,C 180,E1 -14603.348,E2 -14603.348} C_VEL
LIN {X 0,Y 335.962,Z 582.26,A -85,B 0,C 180,E1 -14605.266,E2 -14605.266} C_VEL
LIN {X 0,Y 335.142,Z 586.345,A -85,B 0,C 180,E1 -14607.474,E2 -14607.474} C_VEL
LIN {X 0,Y 334.685,Z 588.181,A -85,B 0,C 180,E1 -14608.88,E2 -14608.88} C_VEL
LIN {X 0,Y 334.291,Z 589.577,A -85,B 0,C 180,E1 -14610.461,E2 -14610.461} C_VEL
LIN {X 0,Y 333.957,Z 590.334,A -85,B 0,C 180,E1 -14612.67,E2 -14612.67} C_VEL
LIN {X 0,Y 333.804,Z 589.811,A -85,B 0,C 180,E1 -14614.803,E2 -14614.803} C_VEL
LIN {X 0,Y 333.826,Z 588.132,A -85,B 0,C 180,E1 -14616.868,E2 -14616.868} C_VEL
LIN {X 0,Y 334.083,Z 584.929,A -85,B 0,C 180,E1 -14619.132,E2 -14619.132} C_VEL
LIN {X 0,Y 334.643,Z 579.931,A -85,B 0,C 180,E1 -14621.461,E2 -14621.461} C_VEL
LIN {X 0,Y 335.147,Z 575.021,A -85,B 0,C 180,E1 -14623.197,E2 -14623.197} C_VEL
LIN {X 0,Y 335.726,Z 569.134,A -85,B 0,C 180,E1 -14624.882,E2 -14624.882} C_VEL
LIN {X 0,Y 336.591,Z 561.641,A -85,B 0,C 180,E1 -14626.624,E2 -14626.624} C_VEL
LIN {X 0,Y 337.453,Z 553.29,A -85,B 0,C 180,E1 -14628.206,E2 -14628.206} C_VEL
LIN {X 0,Y 338.456,Z 542.685,A -85,B 0,C 180,E1 -14629.834,E2 -14629.834} C_VEL
LIN {X 0,Y 339.378,Z 532.028,A -85,B 0,C 180,E1 -14631.153,E2 -14631.153} C_VEL
LIN {X 0,Y 339.6,Z 527.664,A -85,B 0,C 180,E1 -14631.621,E2 -14631.621} C_VEL
LIN {X 0,Y 336.455,Z 516.263,A -85,B 0,C 180,E1 -14632.866,E2 -14632.866} C_VEL
LIN {X 0,Y 333.686,Z 506.92,A -85,B 0,C 180,E1 -14633.745,E2 -14633.745} C_VEL
LIN {X 0,Y 333.648,Z 506.927,A -85,B 0,C 180,E1 -14637.413,E2 -14637.413} C_VEL
LIN {X 0,Y 333.716,Z 506.915,A -85,B 0,C 180,E1 -14641.028,E2 -14641.028} C_VEL
LIN {X 0,Y 333.74,Z 506.912,A -85,B 0,C 180,E1 -14643.754,E2 -14643.754} C_VEL
LIN {X 0,Y 333.661,Z 506.922,A -85,B 0,C 180,E1 -14647.719,E2 -14647.719} C_VEL
LIN {X 0,Y 333.746,Z 506.913,A -85,B 0,C 180,E1 -14651.586,E2 -14651.586} C_VEL
LIN {X 0,Y 333.813,Z 506.904,A -85,B 0,C 180,E1 -14655.577,E2 -14655.577} C_VEL
LIN {X 0,Y 333.823,Z 506.903,A -85,B 0,C 180,E1 -14659.077,E2 -14659.077} C_VEL
LIN {X 0,Y 333.962,Z 506.883,A -85,B 0,C 180,E1 -14662.746,E2 -14662.746} C_VEL
LIN {X 0,Y 333.806,Z 506.906,A -85,B 0,C 180,E1 -14665.169,E2 -14665.169} C_VEL
LIN {X 0,Y 334.11,Z 506.867,A -85,B 0,C 180,E1 -14667.589,E2 -14667.589} C_VEL
LIN {X 0,Y 334.174,Z 506.856,A -85,B 0,C 180,E1 -14670,E2 -14670} C_VEL
LIN {X 0,Y 334.106,Z 506.864,A -85,B 0,C 180,E1 -14672.411,E2 -14672.411} C_VEL
LIN {X 0,Y 333.996,Z 506.878,A -85,B 0,C 180,E1 -14676.039,E2 -14676.039} C_VEL
LIN {X 0,Y 333.825,Z 506.901,A -85,B 0,C 180,E1 -14679.696,E2 -14679.696} C_VEL
LIN {X 0,Y 333.801,Z 506.906,A -85,B 0,C 180,E1 -14683.391,E2 -14683.391} C_VEL
LIN {X 0,Y 333.724,Z 506.917,A -85,B 0,C 180,E1 -14687.147,E2 -14687.147} C_VEL
LIN {X 0,Y 333.728,Z 506.913,A -85,B 0,C 180,E1 -14689.691,E2 -14689.691} C_VEL
LIN {X 0,Y 333.696,Z 506.915,A -85,B 0,C 180,E1 -14692.278,E2 -14692.278} C_VEL
LIN {X 0,Y 333.71,Z 506.919,A -85,B 0,C 180,E1 -14695.096,E2 -14695.096} C_VEL
LIN {X 0,Y 333.674,Z 506.922,A -85,B 0,C 180,E1 -14698.976,E2 -14698.976} C_VEL
LIN {X 0,Y 333.647,Z 506.922,A -85,B 0,C 180,E1 -14702.587,E2 -14702.587} C_VEL
LIN {X 0,Y 333.678,Z 506.918,A -85,B 0,C 180,E1 -14706.139,E2 -14706.139} C_VEL
LIN {X 0,Y 333.623,Z 506.93,A -85,B 0,C 180,E1 -14709.196,E2 -14709.196} C_VEL
LIN {X 0,Y 333.631,Z 506.924,A -85,B 0,C 180,E1 -14712.499,E2 -14712.499} C_VEL
LIN {X 0,Y 333.599,Z 506.928,A -85,B 0,C 180,E1 -14715.955,E2 -14715.955} C_VEL
LIN {X 0,Y 333.649,Z 506.925,A -85,B 0,C 180,E1 -14719.315,E2 -14719.315} C_VEL
LIN {X 0,Y 333.667,Z 506.924,A -85,B 0,C 180,E1 -14723.168,E2 -14723.168} C_VEL
LIN {X 0,Y 333.677,Z 506.921,A -85,B 0,C 180,E1 -14725.341,E2 -14725.341} C_VEL
LIN {X 0,Y 333.705,Z 506.915,A -85,B 0,C 180,E1 -14729.71,E2 -14729.71} C_VEL
LIN {X 0,Y 333.719,Z 506.91,A -85,B 0,C 180,E1 -14733.284,E2 -14733.284} C_VEL
LIN {X 0,Y 333.067,Z 506.995,A -85,B 0,C 180,E1 -14734.29,E2 -14734.29} C_VEL
LIN {X 0,Y 330.209,Z 507.358,A -85,B 0,C 180,E1 -14735.927,E2 -14735.927} C_VEL
LIN {X 0,Y 327.768,Z 507.662,A -85,B 0,C 180,E1 -14737.253,E2 -14737.253} C_VEL
LIN {X 0,Y 326.71,Z 507.789,A -85,B 0,C 180,E1 -14738.279,E2 -14738.279} C_VEL
LIN {X 0,Y 326.619,Z 507.798,A -85,B 0,C 180,E1 -14738.627,E2 -14738.627} C_VEL
LIN {X 0,Y 326.747,Z 507.785,A -85,B 0,C 180,E1 -14741.177,E2 -14741.177} C_VEL
LIN {X 0,Y 326.765,Z 507.78,A -85,B 0,C 180,E1 -14745.433,E2 -14745.433} C_VEL
LIN {X 0,Y 326.761,Z 507.784,A -85,B 0,C 180,E1 -14748.838,E2 -14748.838} C_VEL
LIN {X 0,Y 326.924,Z 507.761,A -85,B 0,C 180,E1 -14752.589,E2 -14752.589} C_VEL
LIN {X 0,Y 326.768,Z 507.783,A -85,B 0,C 180,E1 -14755.064,E2 -14755.064} C_VEL
LIN {X 0,Y 327.045,Z 507.745,A -85,B 0,C 180,E1 -14757.536,E2 -14757.536} C_VEL
LIN {X 0,Y 327.161,Z 507.729,A -85,B 0,C 180,E1 -14760,E2 -14760} C_VEL
LIN {X 0,Y 327.034,Z 507.747,A -85,B 0,C 180,E1 -14762.463,E2 -14762.463} C_VEL
LIN {X 0,Y 326.946,Z 507.756,A -85,B 0,C 180,E1 -14766.17,E2 -14766.17} C_VEL
LIN {X 0,Y 326.807,Z 507.773,A -85,B 0,C 180,E1 -14769.906,E2 -14769.906} C_VEL
LIN {X 0,Y 326.762,Z 507.779,A -85,B 0,C 180,E1 -14773.685,E2 -14773.685} C_VEL
LIN {X 0,Y 326.665,Z 507.792,A -85,B 0,C 180,E1 -14777.53,E2 -14777.53} C_VEL
LIN {X 0,Y 326.632,Z 507.796,A -85,B 0,C 180,E1 -14780.137,E2 -14780.137} C_VEL
LIN {X 0,Y 326.642,Z 507.794,A -85,B 0,C 180,E1 -14784.129,E2 -14784.129} C_VEL
LIN {X 0,Y 326.622,Z 507.798,A -85,B 0,C 180,E1 -14788.254,E2 -14788.254} C_VEL
LIN {X 0,Y 326.574,Z 507.805,A -85,B 0,C 180,E1 -14791.097,E2 -14791.097} C_VEL
LIN {X 0,Y 326.608,Z 507.798,A -85,B 0,C 180,E1 -14794.019,E2 -14794.019} C_VEL
LIN {X 0,Y 326.628,Z 507.797,A -85,B 0,C 180,E1 -14797.238,E2 -14797.238} C_VEL
LIN {X 0,Y 326.586,Z 507.806,A -85,B 0,C 180,E1 -14801.133,E2 -14801.133} C_VEL
LIN {X 0,Y 326.622,Z 507.802,A -85,B 0,C 180,E1 -14802.305,E2 -14802.305} C_VEL
LIN {X 0,Y 328.194,Z 515.701,A -85,B 0,C 180,E1 -14805.838,E2 -14805.838} C_VEL
LIN {X 0,Y 330.114,Z 525.632,A -85,B 0,C 180,E1 -14810.034,E2 -14810.034} C_VEL
LIN {X 0,Y 330.914,Z 530.462,A -85,B 0,C 180,E1 -14811.982,E2 -14811.982} C_VEL
LIN {X 0,Y 330.181,Z 536.943,A -85,B 0,C 180,E1 -14814.419,E2 -14814.419} C_VEL
LIN {X 0,Y 328.846,Z 547.575,A -85,B 0,C 180,E1 -14818.319,E2 -14818.319} C_VEL
LIN {X 0,Y 327.559,Z 559.318,A -85,B 0,C 180,E1 -14822.529,E2 -14822.529} C_VEL
LIN {X 0,Y 326.745,Z 568.709,A -85,B 0,C 180,E1 -14825.879,E2 -14825.879} C_VEL
LIN {X 0,Y 326.219,Z 576.44,A -85,B 0,C 180,E1 -14828.599,E2 -14828.599} C_VEL
LIN {X 0,Y 327.74,Z 591.29,A -85,B 0,C 180,E1 -14829.279,E2 -14829.279} C_VEL
LIN {X 0,Y 328.798,Z 604.63,A -85,B 0,C 180,E1 -14830.135,E2 -14830.135} C_VEL
LIN {X 0,Y 329.326,Z 617.314,A -85,B 0,C 180,E1 -14831.197,E2 -14831.197} C_VEL
LIN {X 0,Y 329.505,Z 629.355,A -85,B 0,C 180,E1 -14832.466,E2 -14832.466} C_VEL
LIN {X 0,Y 328.397,Z 640.035,A -85,B 0,C 180,E1 -14833.847,E2 -14833.847} C_VEL
LIN {X 0,Y 327.267,Z 649.685,A -85,B 0,C 180,E1 -14835.385,E2 -14835.385} C_VEL
LIN {X 0,Y 326.59,Z 657.674,A -85,B 0,C 180,E1 -14836.941,E2 -14836.941} C_VEL
LIN {X 0,Y 325.992,Z 665.485,A -85,B 0,C 180,E1 -14838.812,E2 -14838.812} C_VEL
LIN {X 0,Y 325.748,Z 671.75,A -85,B 0,C 180,E1 -14840.688,E2 -14840.688} C_VEL
LIN {X 0,Y 325.753,Z 677.59,A -85,B 0,C 180,E1 -14842.947,E2 -14842.947} C_VEL
LIN {X 0,Y 325.997,Z 681.515,A -85,B 0,C 180,E1 -14845.053,E2 -14845.053} C_VEL
LIN {X 0,Y 326.108,Z 683.161,A -85,B 0,C 180,E1 -14846.293,E2 -14846.293} C_VEL
LIN {X 0,Y 326.198,Z 684.367,A -85,B 0,C 180,E1 -14847.53,E2 -14847.53} C_VEL
LIN {X 0,Y 326.291,Z 685.147,A -85,B 0,C 180,E1 -14848.766,E2 -14848.766} C_VEL
LIN {X 0,Y 326.537,Z 685.485,A -85,B 0,C 180,E1 -14850,E2 -14850} C_VEL
LIN {X 0,Y 326.142,Z 684.745,A -85,B 0,C 180,E1 -14852.47,E2 -14852.47} C_VEL
LIN {X 0,Y 326.06,Z 683.77,A -85,B 0,C 180,E1 -14853.708,E2 -14853.708} C_VEL
LIN {X 0,Y 325.904,Z 682.321,A -85,B 0,C 180,E1 -14854.949,E2 -14854.949} C_VEL
LIN {X 0,Y 325.681,Z 679.078,A -85,B 0,C 180,E1 -14856.949,E2 -14856.949} C_VEL
LIN {X 0,Y 325.627,Z 673.712,A -85,B 0,C 180,E1 -14859.316,E2 -14859.316} C_VEL
LIN {X 0,Y 325.998,Z 667.145,A -85,B 0,C 180,E1 -14861.503,E2 -14861.503} C_VEL
LIN {X 0,Y 326.854,Z 658.752,A -85,B 0,C 180,E1 -14863.682,E2 -14863.682} C_VEL
LIN {X 0,Y 327.616,Z 651.61,A -85,B 0,C 180,E1 -14865.204,E2 -14865.204} C_VEL
LIN {X 0,Y 328.918,Z 642.823,A -85,B 0,C 180,E1 -14866.766,E2 -14866.766} C_VEL
LIN {X 0,Y 330.547,Z 632.429,A -85,B 0,C 180,E1 -14868.277,E2 -14868.277} C_VEL
LIN {X 0,Y 331.022,Z 620.871,A -85,B 0,C 180,E1 -14869.697,E2 -14869.697} C_VEL
LIN {X 0,Y 331.302,Z 608.759,A -85,B 0,C 180,E1 -14870.919,E2 -14870.919} C_VEL
LIN {X 0,Y 330.836,Z 596.458,A -85,B 0,C 180,E1 -14871.965,E2 -14871.965} C_VEL
LIN {X 0,Y 329.367,Z 583.799,A -85,B 0,C 180,E1 -14872.886,E2 -14872.886} C_VEL
LIN {X 0,Y 326.92,Z 571.044,A -85,B 0,C 180,E1 -14873.687,E2 -14873.687} C_VEL
LIN {X 0,Y 326.565,Z 568.403,A -85,B 0,C 180,E1 -14873.862,E2 -14873.862} C_VEL
LIN {X 0,Y 327.405,Z 558.11,A -85,B 0,C 180,E1 -14877.485,E2 -14877.485} C_VEL
LIN {X 0,Y 328.57,Z 546.708,A -85,B 0,C 180,E1 -14881.649,E2 -14881.649} C_VEL
LIN {X 0,Y 329.946,Z 536.452,A -85,B 0,C 180,E1 -14885.569,E2 -14885.569} C_VEL
LIN {X 0,Y 330.831,Z 530.308,A -85,B 0,C 180,E1 -14888.029,E2 -14888.029} C_VEL
LIN {X 0,Y 330.065,Z 524.658,A -85,B 0,C 180,E1 -14890.588,E2 -14890.588} C_VEL
LIN {X 0,Y 328.656,Z 517.348,A -85,B 0,C 180,E1 -14894.246,E2 -14894.246} C_VEL
LIN {X 0,Y 327.421,Z 511.487,A -85,B 0,C 180,E1 -14897.54,E2 -14897.54} C_VEL
LIN {X 0,Y 326.583,Z 507.805,A -85,B 0,C 180,E1 -14899.926,E2 -14899.926} C_VEL
LIN {X 0,Y 326.632,Z 507.8,A -85,B 0,C 180,E1 -14902.954,E2 -14902.954} C_VEL
LIN {X 0,Y 326.609,Z 507.798,A -85,B 0,C 180,E1 -14905.981,E2 -14905.981} C_VEL
LIN {X 0,Y 326.663,Z 507.789,A -85,B 0,C 180,E1 -14910.341,E2 -14910.341} C_VEL
LIN {X 0,Y 326.693,Z 507.789,A -85,B 0,C 180,E1 -14914.517,E2 -14914.517} C_VEL
LIN {X 0,Y 326.648,Z 507.791,A -85,B 0,C 180,E1 -14918.546,E2 -14918.546} C_VEL
LIN {X 0,Y 326.747,Z 507.782,A -85,B 0,C 180,E1 -14921.178,E2 -14921.178} C_VEL
LIN {X 0,Y 326.766,Z 507.775,A -85,B 0,C 180,E1 -14925.433,E2 -14925.433} C_VEL
LIN {X 0,Y 326.773,Z 507.775,A -85,B 0,C 180,E1 -14928.839,E2 -14928.839} C_VEL
LIN {X 0,Y 326.983,Z 507.751,A -85,B 0,C 180,E1 -14932.591,E2 -14932.591} C_VEL
LIN {X 0,Y 326.77,Z 507.774,A -85,B 0,C 180,E1 -14935.065,E2 -14935.065} C_VEL
LIN {X 0,Y 327.038,Z 507.748,A -85,B 0,C 180,E1 -14937.537,E2 -14937.537} C_VEL
LIN {X 0,Y 327.182,Z 507.73,A -85,B 0,C 180,E1 -14940,E2 -14940} C_VEL
LIN {X 0,Y 327.049,Z 507.748,A -85,B 0,C 180,E1 -14942.464,E2 -14942.464} C_VEL
LIN {X 0,Y 326.926,Z 507.756,A -85,B 0,C 180,E1 -14946.508,E2 -14946.508} C_VEL
LIN {X 0,Y 326.809,Z 507.779,A -85,B 0,C 180,E1 -14949.907,E2 -14949.907} C_VEL
LIN {X 0,Y 326.808,Z 507.774,A -85,B 0,C 180,E1 -14951.042,E2 -14951.042} C_VEL
LIN {X 0,Y 327.501,Z 510.12,A -85,B 0,C 180,E1 -14951.293,E2 -14951.293} C_VEL
LIN {X 0,Y 331.84,Z 520.008,A -85,B 0,C 180,E1 -14952.538,E2 -14952.538} C_VEL
LIN {X 0,Y 335.254,Z 529.959,A -85,B 0,C 180,E1 -14953.866,E2 -14953.866} C_VEL
LIN {X 0,Y 336.758,Z 535.453,A -85,B 0,C 180,E1 -14954.658,E2 -14954.658} C_VEL
LIN {X 0,Y 335.865,Z 544.435,A -85,B 0,C 180,E1 -14955.785,E2 -14955.785} C_VEL
LIN {X 0,Y 334.442,Z 554.26,A -85,B 0,C 180,E1 -14957.267,E2 -14957.267} C_VEL
LIN {X 0,Y 333.169,Z 562.172,A -85,B 0,C 180,E1 -14958.733,E2 -14958.733} C_VEL
LIN {X 0,Y 331.84,Z 569.677,A -85,B 0,C 180,E1 -14960.424,E2 -14960.424} C_VEL
LIN {X 0,Y 330.468,Z 576.923,A -85,B 0,C 180,E1 -14962.508,E2 -14962.508} C_VEL
LIN {X 0,Y 329.329,Z 582.487,A -85,B 0,C 180,E1 -14964.591,E2 -14964.591} C_VEL
LIN {X 0,Y 328.414,Z 586.618,A -85,B 0,C 180,E1 -14966.706,E2 -14966.706} C_VEL
LIN {X 0,Y 327.82,Z 589.06,A -85,B 0,C 180,E1 -14968.479,E2 -14968.479} C_VEL
LIN {X 0,Y 327.217,Z 590.906,A -85,B 0,C 180,E1 -14970.781,E2 -14970.781} C_VEL
LIN {X 0,Y 326.906,Z 591.383,A -85,B 0,C 180,E1 -14973.023,E2 -14973.023} C_VEL
LIN {X 0,Y 326.781,Z 590.395,A -85,B 0,C 180,E1 -14975.499,E2 -14975.499} C_VEL
LIN {X 0,Y 326.83,Z 588.694,A -85,B 0,C 180,E1 -14977.284,E2 -14977.284} C_VEL
LIN {X 0,Y 327.078,Z 585.643,A -85,B 0,C 180,E1 -14979.327,E2 -14979.327} C_VEL
LIN {X 0,Y 327.675,Z 580.602,A -85,B 0,C 180,E1 -14981.675,E2 -14981.675} C_VEL
LIN {X 0,Y 328.28,Z 574.919,A -85,B 0,C 180,E1 -14983.665,E2 -14983.665} C_VEL
LIN {X 0,Y 329.129,Z 567.218,A -85,B 0,C 180,E1 -14985.755,E2 -14985.755} C_VEL
LIN {X 0,Y 330.05,Z 559.203,A -85,B 0,C 180,E1 -14987.5,E2 -14987.5} C_VEL
LIN {X 0,Y 331.048,Z 549.339,A -85,B 0,C 180,E1 -14989.232,E2 -14989.232} C_VEL
LIN {X 0,Y 332.094,Z 538.112,A -85,B 0,C 180,E1 -14990.815,E2 -14990.815} C_VEL
LIN {X 0,Y 332.782,Z 529.867,A -85,B 0,C 180,E1 -14991.762,E2 -14991.762} C_VEL
LIN {X 0,Y 330.149,Z 519.674,A -85,B 0,C 180,E1 -14992.934,E2 -14992.934} C_VEL
LIN {X 0,Y 326.638,Z 507.795,A -85,B 0,C 180,E1 -14994.104,E2 -14994.104} C_VEL
LIN {X 0,Y 326.612,Z 507.803,A -85,B 0,C 180,E1 -14997.456,E2 -14997.456} C_VEL
LIN {X 0,Y 326.665,Z 507.791,A -85,B 0,C 180,E1 -15000.341,E2 -15000.341} C_VEL
LIN {X 0,Y 326.695,Z 507.787,A -85,B 0,C 180,E1 -15004.516,E2 -15004.516} C_VEL
LIN {X 0,Y 326.623,Z 507.796,A -85,B 0,C 180,E1 -15008.543,E2 -15008.543} C_VEL
LIN {X 0,Y 326.712,Z 507.789,A -85,B 0,C 180,E1 -15011.175,E2 -15011.175} C_VEL
LIN {X 0,Y 326.768,Z 507.783,A -85,B 0,C 180,E1 -15015.433,E2 -15015.433} C_VEL
LIN {X 0,Y 326.764,Z 507.78,A -85,B 0,C 180,E1 -15018.839,E2 -15018.839} C_VEL
LIN {X 0,Y 326.919,Z 507.76,A -85,B 0,C 180,E1 -15022.589,E2 -15022.589} C_VEL
LIN {X 0,Y 326.772,Z 507.781,A -85,B 0,C 180,E1 -15025.065,E2 -15025.065} C_VEL
LIN {X 0,Y 327.05,Z 507.747,A -85,B 0,C 180,E1 -15027.537,E2 -15027.537} C_VEL
LIN {X 0,Y 327.129,Z 507.734,A -85,B 0,C 180,E1 -15030,E2 -15030} C_VEL
LIN {X 0,Y 327.046,Z 507.744,A -85,B 0,C 180,E1 -15032.463,E2 -15032.463} C_VEL
LIN {X 0,Y 326.95,Z 507.756,A -85,B 0,C 180,E1 -15036.17,E2 -15036.17} C_VEL
LIN {X 0,Y 326.788,Z 507.776,A -85,B 0,C 180,E1 -15039.907,E2 -15039.907} C_VEL
LIN {X 0,Y 326.764,Z 507.78,A -85,B 0,C 180,E1 -15043.685,E2 -15043.685} C_VEL
LIN {X 0,Y 326.669,Z 507.793,A -85,B 0,C 180,E1 -15047.529,E2 -15047.529} C_VEL
LIN {X 0,Y 326.661,Z 507.791,A -85,B 0,C 180,E1 -15050.135,E2 -15050.135} C_VEL
LIN {X 0,Y 326.65,Z 507.793,A -85,B 0,C 180,E1 -15054.129,E2 -15054.129} C_VEL
LIN {X 0,Y 326.631,Z 507.795,A -85,B 0,C 180,E1 -15058.253,E2 -15058.253} C_VEL
LIN {X 0,Y 326.579,Z 507.807,A -85,B 0,C 180,E1 -15061.097,E2 -15061.097} C_VEL
LIN {X 0,Y 326.61,Z 507.798,A -85,B 0,C 180,E1 -15064.019,E2 -15064.019} C_VEL
LIN {X 0,Y 326.626,Z 507.801,A -85,B 0,C 180,E1 -15067.237,E2 -15067.237} C_VEL
LIN {X 0,Y 326.547,Z 507.812,A -85,B 0,C 180,E1 -15071.124,E2 -15071.124} C_VEL
LIN {X 0,Y 326.563,Z 507.806,A -85,B 0,C 180,E1 -15073.525,E2 -15073.525} C_VEL
LIN {X 0,Y 326.578,Z 507.807,A -85,B 0,C 180,E1 -15077.028,E2 -15077.028} C_VEL
LIN {X 0,Y 326.613,Z 507.8,A -85,B 0,C 180,E1 -15080.773,E2 -15080.773} C_VEL
LIN {X 0,Y 326.615,Z 507.798,A -85,B 0,C 180,E1 -15084.48,E2 -15084.48} C_VEL
LIN {X 0,Y 326.61,Z 507.8,A -85,B 0,C 180,E1 -15087.455,E2 -15087.455} C_VEL
LIN {X 0,Y 326.663,Z 507.792,A -85,B 0,C 180,E1 -15090.341,E2 -15090.341} C_VEL
LIN {X 0,Y 326.692,Z 507.789,A -85,B 0,C 180,E1 -15094.516,E2 -15094.516} C_VEL
LIN {X 0,Y 326.619,Z 507.798,A -85,B 0,C 180,E1 -15098.627,E2 -15098.627} C_VEL
LIN {X 0,Y 325.944,Z 507.882,A -85,B 0,C 180,E1 -15099.657,E2 -15099.657} C_VEL
LIN {X 0,Y 323.116,Z 508.236,A -85,B 0,C 180,E1 -15101.335,E2 -15101.335} C_VEL
LIN {X 0,Y 320.741,Z 508.532,A -85,B 0,C 180,E1 -15102.694,E2 -15102.694} C_VEL
LIN {X 0,Y 319.741,Z 508.654,A -85,B 0,C 180,E1 -15103.745,E2 -15103.745} C_VEL
LIN {X 0,Y 319.669,Z 508.662,A -85,B 0,C 180,E1 -15104.101,E2 -15104.101} C_VEL
LIN {X 0,Y 319.684,Z 508.663,A -85,B 0,C 180,E1 -15107.3,E2 -15107.3} C_VEL
LIN {X 0,Y 319.828,Z 508.644,A -85,B 0,C 180,E1 -15111.435,E2 -15111.435} C_VEL
LIN {X 0,Y 319.911,Z 508.633,A -85,B 0,C 180,E1 -15113.693,E2 -15113.693} C_VEL
LIN {X 0,Y 319.988,Z 508.624,A -85,B 0,C 180,E1 -15117.482,E2 -15117.482} C_VEL
LIN {X 0,Y 320.113,Z 508.607,A -85,B 0,C 180,E1 -15120,E2 -15120} C_VEL
LIN {X 0,Y 319.977,Z 508.626,A -85,B 0,C 180,E1 -15122.517,E2 -15122.517} C_VEL
LIN {X 0,Y 319.903,Z 508.634,A -85,B 0,C 180,E1 -15126.306,E2 -15126.306} C_VEL
LIN {X 0,Y 319.755,Z 508.652,A -85,B 0,C 180,E1 -15130.127,E2 -15130.127} C_VEL
LIN {X 0,Y 319.734,Z 508.654,A -85,B 0,C 180,E1 -15133.992,E2 -15133.992} C_VEL
LIN {X 0,Y 319.625,Z 508.668,A -85,B 0,C 180,E1 -15137.929,E2 -15137.929} C_VEL
LIN {X 0,Y 319.568,Z 508.675,A -85,B 0,C 180,E1 -15141.954,E2 -15141.954} C_VEL
LIN {X 0,Y 319.574,Z 508.675,A -85,B 0,C 180,E1 -15146.093,E2 -15146.093} C_VEL
LIN {X 0,Y 319.553,Z 508.681,A -85,B 0,C 180,E1 -15148.937,E2 -15148.937} C_VEL
LIN {X 0,Y 319.525,Z 508.681,A -85,B 0,C 180,E1 -15151.862,E2 -15151.862} C_VEL
LIN {X 0,Y 319.58,Z 508.674,A -85,B 0,C 180,E1 -15155.543,E2 -15155.543} C_VEL
LIN {X 0,Y 319.557,Z 508.677,A -85,B 0,C 180,E1 -15158.01,E2 -15158.01} C_VEL
LIN {X 0,Y 319.592,Z 508.737,A -85,B 0,C 180,E1 -15161.951,E2 -15161.951} C_VEL
LIN {X 0,Y 321.121,Z 516.574,A -85,B 0,C 180,E1 -15165.545,E2 -15165.545} C_VEL
LIN {X 0,Y 322.757,Z 525.002,A -85,B 0,C 180,E1 -15169.213,E2 -15169.213} C_VEL
LIN {X 0,Y 323.894,Z 531.75,A -85,B 0,C 180,E1 -15172.006,E2 -15172.006} C_VEL
LIN {X 0,Y 322.982,Z 539.026,A -85,B 0,C 180,E1 -15174.786,E2 -15174.786} C_VEL
LIN {X 0,Y 321.723,Z 548.707,A -85,B 0,C 180,E1 -15178.425,E2 -15178.425} C_VEL
LIN {X 0,Y 320.443,Z 559.973,A -85,B 0,C 180,E1 -15182.576,E2 -15182.576} C_VEL
LIN {X 0,Y 319.63,Z 569.385,A -85,B 0,C 180,E1 -15185.998,E2 -15185.998} C_VEL
LIN {X 0,Y 319.197,Z 575.579,A -85,B 0,C 180,E1 -15188.231,E2 -15188.231} C_VEL
LIN {X 0,Y 320.687,Z 590.135,A -85,B 0,C 180,E1 -15188.906,E2 -15188.906} C_VEL
LIN {X 0,Y 321.643,Z 602.495,A -85,B 0,C 180,E1 -15189.704,E2 -15189.704} C_VEL
LIN {X 0,Y 322.212,Z 615.391,A -85,B 0,C 180,E1 -15190.789,E2 -15190.789} C_VEL
LIN {X 0,Y 322.412,Z 627.476,A -85,B 0,C 180,E1 -15192.067,E2 -15192.067} C_VEL
LIN {X 0,Y 322.105,Z 633.878,A -85,B 0,C 180,E1 -15192.869,E2 -15192.869} C_VEL
LIN {X 0,Y 321.051,Z 642.951,A -85,B 0,C 180,E1 -15194.185,E2 -15194.185} C_VEL
LIN {X 0,Y 319.956,Z 651.616,A -85,B 0,C 180,E1 -15195.708,E2 -15195.708} C_VEL
LIN {X 0,Y 319.255,Z 660.405,A -85,B 0,C 180,E1 -15197.606,E2 -15197.606} C_VEL
LIN {X 0,Y 318.826,Z 667.484,A -85,B 0,C 180,E1 -15199.522,E2 -15199.522} C_VEL
LIN {X 0,Y 318.671,Z 673.945,A -85,B 0,C 180,E1 -15201.758,E2 -15201.758} C_VEL
LIN {X 0,Y 318.737,Z 678.149,A -85,B 0,C 180,E1 -15203.671,E2 -15203.671} C_VEL
LIN {X 0,Y 318.941,Z 680.357,A -85,B 0,C 180,E1 -15204.943,E2 -15204.943} C_VEL
LIN {X 0,Y 319.06,Z 682.029,A -85,B 0,C 180,E1 -15206.211,E2 -15206.211} C_VEL
LIN {X 0,Y 319.163,Z 683.257,A -85,B 0,C 180,E1 -15207.476,E2 -15207.476} C_VEL
LIN {X 0,Y 319.29,Z 684.061,A -85,B 0,C 180,E1 -15208.739,E2 -15208.739} C_VEL
LIN {X 0,Y 319.509,Z 684.434,A -85,B 0,C 180,E1 -15210,E2 -15210} C_VEL
LIN {X 0,Y 319.097,Z 683.729,A -85,B 0,C 180,E1 -15212.525,E2 -15212.525} C_VEL
LIN {X 0,Y 319.011,Z 682.77,A -85,B 0,C 180,E1 -15213.79,E2 -15213.79} C_VEL
LIN {X 0,Y 318.828,Z 681.357,A -85,B 0,C 180,E1 -15215.059,E2 -15215.059} C_VEL
LIN {X 0,Y 318.608,Z 678.421,A -85,B 0,C 180,E1 -15216.96,E2 -15216.96} C_VEL
LIN {X 0,Y 318.531,Z 674.412,A -85,B 0,C 180,E1 -15218.885,E2 -15218.885} C_VEL
LIN {X 0,Y 318.707,Z 669.318,A -85,B 0,C 180,E1 -15220.804,E2 -15220.804} C_VEL
LIN {X 0,Y 319.423,Z 661.826,A -85,B 0,C 180,E1 -15223.034,E2 -15223.034} C_VEL
LIN {X 0,Y 320.117,Z 655.836,A -85,B 0,C 180,E1 -15224.504,E2 -15224.504} C_VEL
LIN {X 0,Y 321.065,Z 649.268,A -85,B 0,C 180,E1 -15225.88,E2 -15225.88} C_VEL
LIN {X 0,Y 322.582,Z 639.415,A -85,B 0,C 180,E1 -15227.596,E2 -15227.596} C_VEL
LIN {X 0,Y 323.707,Z 632.035,A -85,B 0,C 180,E1 -15228.678,E2 -15228.678} C_VEL
LIN {X 0,Y 324.273,Z 620.717,A -85,B 0,C 180,E1 -15230.125,E2 -15230.125} C_VEL
LIN {X 0,Y 324.655,Z 608.282,A -85,B 0,C 180,E1 -15231.433,E2 -15231.433} C_VEL
LIN {X 0,Y 324.123,Z 595.425,A -85,B 0,C 180,E1 -15232.576,E2 -15232.576} C_VEL
LIN {X 0,Y 322.493,Z 582.422,A -85,B 0,C 180,E1 -15233.563,E2 -15233.563} C_VEL
LIN {X 0,Y 320.01,Z 569.734,A -85,B 0,C 180,E1 -15234.411,E2 -15234.411} C_VEL
LIN {X 0,Y 319.629,Z 567.111,A -85,B 0,C 180,E1 -15234.58,E2 -15234.58} C_VEL
LIN {X 0,Y 320.712,Z 555.463,A -85,B 0,C 180,E1 -15238.823,E2 -15238.823} C_VEL
LIN {X 0,Y 322.015,Z 544.275,A -85,B 0,C 180,E1 -15243.068,E2 -15243.068} C_VEL
LIN {X 0,Y 323.764,Z 533.36,A -85,B 0,C 180,E1 -15247.431,E2 -15247.431} C_VEL
LIN {X 0,Y 323.712,Z 529.737,A -85,B 0,C 180,E1 -15249.022,E2 -15249.022} C_VEL
LIN {X 0,Y 322.562,Z 523.169,A -85,B 0,C 180,E1 -15252.201,E2 -15252.201} C_VEL
LIN {X 0,Y 321.317,Z 516.881,A -85,B 0,C 180,E1 -15255.579,E2 -15255.579} C_VEL
LIN {X 0,Y 320.164,Z 511.513,A -85,B 0,C 180,E1 -15258.812,E2 -15258.812} C_VEL
LIN {X 0,Y 319.592,Z 508.678,A -85,B 0,C 180,E1 -15260.786,E2 -15260.786} C_VEL
LIN {X 0,Y 319.562,Z 508.679,A -85,B 0,C 180,E1 -15265.124,E2 -15265.124} C_VEL
LIN {X 0,Y 319.572,Z 508.676,A -85,B 0,C 180,E1 -15269.058,E2 -15269.058} C_VEL
LIN {X 0,Y 319.611,Z 508.67,A -85,B 0,C 180,E1 -15272.499,E2 -15272.499} C_VEL
LIN {X 0,Y 319.608,Z 508.67,A -85,B 0,C 180,E1 -15275.304,E2 -15275.304} C_VEL
LIN {X 0,Y 319.599,Z 508.673,A -85,B 0,C 180,E1 -15278.048,E2 -15278.048} C_VEL
LIN {X 0,Y 319.692,Z 508.663,A -85,B 0,C 180,E1 -15280.963,E2 -15280.963} C_VEL
LIN {X 0,Y 319.734,Z 508.651,A -85,B 0,C 180,E1 -15285.276,E2 -15285.276} C_VEL
LIN {X 0,Y 319.761,Z 508.655,A -85,B 0,C 180,E1 -15289.873,E2 -15289.873} C_VEL
LIN {X 0,Y 319.937,Z 508.627,A -85,B 0,C 180,E1 -15292.427,E2 -15292.427} C_VEL
LIN {X 0,Y 319.741,Z 508.65,A -85,B 0,C 180,E1 -15294.956,E2 -15294.956} C_VEL
LIN {X 0,Y 319.981,Z 508.627,A -85,B 0,C 180,E1 -15297.483,E2 -15297.483} C_VEL
LIN {X 0,Y 320.134,Z 508.607,A -85,B 0,C 180,E1 -15300,E2 -15300} C_VEL
LIN {X 0,Y 319.992,Z 508.628,A -85,B 0,C 180,E1 -15302.518,E2 -15302.518} C_VEL
LIN {X 0,Y 319.89,Z 508.632,A -85,B 0,C 180,E1 -15306.49,E2 -15306.49} C_VEL
LIN {X 0,Y 319.756,Z 508.658,A -85,B 0,C 180,E1 -15310.287,E2 -15310.287} C_VEL
LIN {X 0,Y 320.544,Z 511.118,A -85,B 0,C 180,E1 -15310.581,E2 -15310.581} C_VEL
LIN {X 0,Y 325.349,Z 521.913,A -85,B 0,C 180,E1 -15312.001,E2 -15312.001} C_VEL
LIN {X 0,Y 328.642,Z 531.642,A -85,B 0,C 180,E1 -15313.37,E2 -15313.37} C_VEL
LIN {X 0,Y 330.345,Z 538.461,A -85,B 0,C 180,E1 -15314.39,E2 -15314.39} C_VEL
LIN {X 0,Y 329.075,Z 548.19,A -85,B 0,C 180,E1 -15315.671,E2 -15315.671} C_VEL
LIN {X 0,Y 327.616,Z 557.386,A -85,B 0,C 180,E1 -15317.156,E2 -15317.156} C_VEL
LIN {X 0,Y 326.106,Z 565.892,A -85,B 0,C 180,E1 -15318.861,E2 -15318.861} C_VEL
LIN {X 0,Y 324.688,Z 573.464,A -85,B 0,C 180,E1 -15320.757,E2 -15320.757} C_VEL
LIN {X 0,Y 323.615,Z 578.546,A -85,B 0,C 180,E1 -15322.337,E2 -15322.337} C_VEL
LIN {X 0,Y 322.424,Z 583.979,A -85,B 0,C 180,E1 -15324.466,E2 -15324.466} C_VEL
LIN {X 0,Y 321.577,Z 587.567,A -85,B 0,C 180,E1 -15326.356,E2 -15326.356} C_VEL
LIN {X 0,Y 320.732,Z 590.654,A -85,B 0,C 180,E1 -15328.777,E2 -15328.777} C_VEL
LIN {X 0,Y 320.163,Z 592.216,A -85,B 0,C 180,E1 -15331.118,E2 -15331.118} C_VEL
LIN {X 0,Y 319.849,Z 592.39,A -85,B 0,C 180,E1 -15333.387,E2 -15333.387} C_VEL
LIN {X 0,Y 319.749,Z 591.33,A -85,B 0,C 180,E1 -15335.585,E2 -15335.585} C_VEL
LIN {X 0,Y 319.857,Z 588.822,A -85,B 0,C 180,E1 -15337.969,E2 -15337.969} C_VEL
LIN {X 0,Y 320.276,Z 584.649,A -85,B 0,C 180,E1 -15340.41,E2 -15340.41} C_VEL
LIN {X 0,Y 320.785,Z 580.382,A -85,B 0,C 180,E1 -15342.236,E2 -15342.236} C_VEL
LIN {X 0,Y 321.53,Z 573.932,A -85,B 0,C 180,E1 -15344.384,E2 -15344.384} C_VEL
LIN {X 0,Y 322.219,Z 567.744,A -85,B 0,C 180,E1 -15346.036,E2 -15346.036} C_VEL
LIN {X 0,Y 323.244,Z 559.19,A -85,B 0,C 180,E1 -15347.899,E2 -15347.899} C_VEL
LIN {X 0,Y 324.2,Z 549.702,A -85,B 0,C 180,E1 -15349.568,E2 -15349.568} C_VEL
LIN {X 0,Y 325.224,Z 539.162,A -85,B 0,C 180,E1 -15351.074,E2 -15351.074} C_VEL
LIN {X 0,Y 325.843,Z 530.732,A -85,B 0,C 180,E1 -15352.069,E2 -15352.069} C_VEL
LIN {X 0,Y 323.142,Z 520.595,A -85,B 0,C 180,E1 -15353.266,E2 -15353.266} C_VEL
LIN {X 0,Y 319.59,Z 508.673,A -85,B 0,C 180,E1 -15354.456,E2 -15354.456} C_VEL
LIN {X 0,Y 319.537,Z 508.68,A -85,B 0,C 180,E1 -15358.138,E2 -15358.138} C_VEL
LIN {X 0,Y 319.621,Z 508.673,A -85,B 0,C 180,E1 -15361.589,E2 -15361.589} C_VEL
LIN {X 0,Y 319.608,Z 508.675,A -85,B 0,C 180,E1 -15365.304,E2 -15365.304} C_VEL
LIN {X 0,Y 319.591,Z 508.678,A -85,B 0,C 180,E1 -15369.399,E2 -15369.399} C_VEL
LIN {X 0,Y 319.629,Z 508.668,A -85,B 0,C 180,E1 -15372.071,E2 -15372.071} C_VEL
LIN {X 0,Y 319.737,Z 508.655,A -85,B 0,C 180,E1 -15376.008,E2 -15376.008} C_VEL
LIN {X 0,Y 319.741,Z 508.655,A -85,B 0,C 180,E1 -15379.872,E2 -15379.872} C_VEL
LIN {X 0,Y 319.907,Z 508.635,A -85,B 0,C 180,E1 -15383.693,E2 -15383.693} C_VEL
LIN {X 0,Y 319.994,Z 508.626,A -85,B 0,C 180,E1 -15387.482,E2 -15387.482} C_VEL
LIN {X 0,Y 320.085,Z 508.611,A -85,B 0,C 180,E1 -15390,E2 -15390} C_VEL
LIN {X 0,Y 319.99,Z 508.623,A -85,B 0,C 180,E1 -15392.517,E2 -15392.517} C_VEL
LIN {X 0,Y 319.906,Z 508.633,A -85,B 0,C 180,E1 -15396.306,E2 -15396.306} C_VEL
LIN {X 0,Y 319.74,Z 508.654,A -85,B 0,C 180,E1 -15400.128,E2 -15400.128} C_VEL
LIN {X 0,Y 319.737,Z 508.654,A -85,B 0,C 180,E1 -15403.992,E2 -15403.992} C_VEL
LIN {X 0,Y 319.629,Z 508.668,A -85,B 0,C 180,E1 -15407.929,E2 -15407.929} C_VEL
LIN {X 0,Y 319.616,Z 508.67,A -85,B 0,C 180,E1 -15410.599,E2 -15410.599} C_VEL
LIN {X 0,Y 319.572,Z 508.679,A -85,B 0,C 180,E1 -15413.319,E2 -15413.319} C_VEL
LIN {X 0,Y 319.583,Z 508.673,A -85,B 0,C 180,E1 -15416.093,E2 -15416.093} C_VEL
LIN {X 0,Y 319.561,Z 508.679,A -85,B 0,C 180,E1 -15418.936,E2 -15418.936} C_VEL
LIN {X 0,Y 319.528,Z 508.68,A -85,B 0,C 180,E1 -15421.862,E2 -15421.862} C_VEL
LIN {X 0,Y 319.583,Z 508.675,A -85,B 0,C 180,E1 -15425.543,E2 -15425.543} C_VEL
LIN {X 0,Y 319.53,Z 508.681,A -85,B 0,C 180,E1 -15429.662,E2 -15429.662} C_VEL
LIN {X 0,Y 319.523,Z 508.683,A -85,B 0,C 180,E1 -15433.46,E2 -15433.46} C_VEL
LIN {X 0,Y 319.556,Z 508.682,A -85,B 0,C 180,E1 -15437.016,E2 -15437.016} C_VEL
LIN {X 0,Y 319.549,Z 508.678,A -85,B 0,C 180,E1 -15440.37,E2 -15440.37} C_VEL
LIN {X 0,Y 319.582,Z 508.674,A -85,B 0,C 180,E1 -15444.457,E2 -15444.457} C_VEL
LIN {X 0,Y 319.535,Z 508.679,A -85,B 0,C 180,E1 -15448.138,E2 -15448.138} C_VEL
LIN {X 0,Y 319.618,Z 508.67,A -85,B 0,C 180,E1 -15451.588,E2 -15451.588} C_VEL
LIN {X 0,Y 319.606,Z 508.673,A -85,B 0,C 180,E1 -15455.304,E2 -15455.304} C_VEL
LIN {X 0,Y 319.604,Z 508.673,A -85,B 0,C 180,E1 -15459.4,E2 -15459.4} C_VEL
LIN {X 0,Y 319.661,Z 508.663,A -85,B 0,C 180,E1 -15462.073,E2 -15462.073} C_VEL
LIN {X 0,Y 319.669,Z 508.662,A -85,B 0,C 180,E1 -15464.101,E2 -15464.101} C_VEL
LIN {X 0,Y 319.032,Z 508.746,A -85,B 0,C 180,E1 -15465.152,E2 -15465.152} C_VEL
LIN {X 0,Y 316.211,Z 509.098,A -85,B 0,C 180,E1 -15466.864,E2 -15466.864} C_VEL
LIN {X 0,Y 313.804,Z 509.397,A -85,B 0,C 180,E1 -15468.251,E2 -15468.251} C_VEL
LIN {X 0,Y 312.771,Z 509.525,A -85,B 0,C 180,E1 -15469.324,E2 -15469.324} C_VEL
LIN {X 0,Y 312.687,Z 509.533,A -85,B 0,C 180,E1 -15469.688,E2 -15469.688} C_VEL
LIN {X 0,Y 312.804,Z 509.518,A -85,B 0,C 180,E1 -15472.252,E2 -15472.252} C_VEL
LIN {X 0,Y 312.705,Z 509.535,A -85,B 0,C 180,E1 -15474.842,E2 -15474.842} C_VEL
LIN {X 0,Y 312.934,Z 509.503,A -85,B 0,C 180,E1 -15477.425,E2 -15477.425} C_VEL
LIN {X 0,Y 313.068,Z 509.485,A -85,B 0,C 180,E1 -15480,E2 -15480} C_VEL
LIN {X 0,Y 312.923,Z 509.505,A -85,B 0,C 180,E1 -15482.574,E2 -15482.574} C_VEL
LIN {X 0,Y 312.844,Z 509.514,A -85,B 0,C 180,E1 -15486.449,E2 -15486.449} C_VEL
LIN {X 0,Y 312.757,Z 509.527,A -85,B 0,C 180,E1 -15489.05,E2 -15489.05} C_VEL
LIN {X 0,Y 312.639,Z 509.542,A -85,B 0,C 180,E1 -15492.991,E2 -15492.991} C_VEL
LIN {X 0,Y 312.623,Z 509.54,A -85,B 0,C 180,E1 -15495.65,E2 -15495.65} C_VEL
LIN {X 0,Y 312.56,Z 509.548,A -85,B 0,C 180,E1 -15499.711,E2 -15499.711} C_VEL
LIN {X 0,Y 312.526,Z 509.557,A -85,B 0,C 180,E1 -15502.78,E2 -15502.78} C_VEL
LIN {X 0,Y 312.534,Z 509.551,A -85,B 0,C 180,E1 -15505.909,E2 -15505.909} C_VEL
LIN {X 0,Y 312.5,Z 509.555,A -85,B 0,C 180,E1 -15509.654,E2 -15509.654} C_VEL
LIN {X 0,Y 312.52,Z 509.553,A -85,B 0,C 180,E1 -15513.689,E2 -15513.689} C_VEL
LIN {X 0,Y 312.526,Z 509.553,A -85,B 0,C 180,E1 -15517.385,E2 -15517.385} C_VEL
LIN {X 0,Y 312.562,Z 509.696,A -85,B 0,C 180,E1 -15521.611,E2 -15521.611} C_VEL
LIN {X 0,Y 314.268,Z 518.406,A -85,B 0,C 180,E1 -15525.694,E2 -15525.694} C_VEL
LIN {X 0,Y 315.773,Z 526.251,A -85,B 0,C 180,E1 -15529.176,E2 -15529.176} C_VEL
LIN {X 0,Y 316.811,Z 531.95,A -85,B 0,C 180,E1 -15531.601,E2 -15531.601} C_VEL
LIN {X 0,Y 316.536,Z 535.881,A -85,B 0,C 180,E1 -15533.168,E2 -15533.168} C_VEL
LIN {X 0,Y 314.939,Z 547.391,A -85,B 0,C 180,E1 -15537.617,E2 -15537.617} C_VEL
LIN {X 0,Y 313.524,Z 558.783,A -85,B 0,C 180,E1 -15541.918,E2 -15541.918} C_VEL
LIN {X 0,Y 312.506,Z 569.992,A -85,B 0,C 180,E1 -15546.121,E2 -15546.121} C_VEL
LIN {X 0,Y 312.15,Z 574.516,A -85,B 0,C 180,E1 -15547.801,E2 -15547.801} C_VEL
LIN {X 0,Y 313.744,Z 589.864,A -85,B 0,C 180,E1 -15548.567,E2 -15548.567} C_VEL
LIN {X 0,Y 314.661,Z 602.241,A -85,B 0,C 180,E1 -15549.404,E2 -15549.404} C_VEL
LIN {X 0,Y 315.157,Z 614.399,A -85,B 0,C 180,E1 -15550.458,E2 -15550.458} C_VEL
LIN {X 0,Y 315.339,Z 625.486,A -85,B 0,C 180,E1 -15551.651,E2 -15551.651} C_VEL
LIN {X 0,Y 315.133,Z 633.277,A -85,B 0,C 180,E1 -15552.645,E2 -15552.645} C_VEL
LIN {X 0,Y 313.987,Z 642.865,A -85,B 0,C 180,E1 -15554.086,E2 -15554.086} C_VEL
LIN {X 0,Y 312.877,Z 651.633,A -85,B 0,C 180,E1 -15555.695,E2 -15555.695} C_VEL
LIN {X 0,Y 312.261,Z 658.944,A -85,B 0,C 180,E1 -15557.324,E2 -15557.324} C_VEL
LIN {X 0,Y 311.773,Z 666.127,A -85,B 0,C 180,E1 -15559.282,E2 -15559.282} C_VEL
LIN {X 0,Y 311.612,Z 672.658,A -85,B 0,C 180,E1 -15561.57,E2 -15561.57} C_VEL
LIN {X 0,Y 311.678,Z 676.923,A -85,B 0,C 180,E1 -15563.527,E2 -15563.527} C_VEL
LIN {X 0,Y 311.889,Z 679.166,A -85,B 0,C 180,E1 -15564.829,E2 -15564.829} C_VEL
LIN {X 0,Y 312.013,Z 680.885,A -85,B 0,C 180,E1 -15566.125,E2 -15566.125} C_VEL
LIN {X 0,Y 312.127,Z 682.138,A -85,B 0,C 180,E1 -15567.419,E2 -15567.419} C_VEL
LIN {X 0,Y 312.285,Z 682.968,A -85,B 0,C 180,E1 -15568.711,E2 -15568.711} C_VEL
LIN {X 0,Y 312.506,Z 683.38,A -85,B 0,C 180,E1 -15570,E2 -15570} C_VEL
LIN {X 0,Y 312.052,Z 682.711,A -85,B 0,C 180,E1 -15572.582,E2 -15572.582} C_VEL
LIN {X 0,Y 311.96,Z 681.769,A -85,B 0,C 180,E1 -15573.876,E2 -15573.876} C_VEL
LIN {X 0,Y 311.756,Z 680.388,A -85,B 0,C 180,E1 -15575.174,E2 -15575.174} C_VEL
LIN {X 0,Y 311.551,Z 677.684,A -85,B 0,C 180,E1 -15576.995,E2 -15576.995} C_VEL
LIN {X 0,Y 311.452,Z 673.521,A -85,B 0,C 180,E1 -15579.089,E2 -15579.089} C_VEL
LIN {X 0,Y 311.674,Z 668.495,A -85,B 0,C 180,E1 -15581.05,E2 -15581.05} C_VEL
LIN {X 0,Y 312.403,Z 661.087,A -85,B 0,C 180,E1 -15583.332,E2 -15583.332} C_VEL
LIN {X 0,Y 313.163,Z 654.262,A -85,B 0,C 180,E1 -15585.041,E2 -15585.041} C_VEL
LIN {X 0,Y 314.712,Z 645.32,A -85,B 0,C 180,E1 -15586.877,E2 -15586.877} C_VEL
LIN {X 0,Y 316.556,Z 634.969,A -85,B 0,C 180,E1 -15588.612,E2 -15588.612} C_VEL
LIN {X 0,Y 317.354,Z 623.289,A -85,B 0,C 180,E1 -15590.245,E2 -15590.245} C_VEL
LIN {X 0,Y 317.95,Z 610.922,A -85,B 0,C 180,E1 -15591.663,E2 -15591.663} C_VEL
LIN {X 0,Y 317.745,Z 599.133,A -85,B 0,C 180,E1 -15592.8,E2 -15592.8} C_VEL
LIN {X 0,Y 316.641,Z 587.273,A -85,B 0,C 180,E1 -15593.809,E2 -15593.809} C_VEL
LIN {X 0,Y 314.27,Z 573.118,A -85,B 0,C 180,E1 -15594.857,E2 -15594.857} C_VEL
LIN {X 0,Y 312.765,Z 565.721,A -85,B 0,C 180,E1 -15595.374,E2 -15595.374} C_VEL
LIN {X 0,Y 313.852,Z 554.723,A -85,B 0,C 180,E1 -15599.515,E2 -15599.515} C_VEL
LIN {X 0,Y 315,Z 545.461,A -85,B 0,C 180,E1 -15603.136,E2 -15603.136} C_VEL
LIN {X 0,Y 316.551,Z 536.142,A -85,B 0,C 180,E1 -15606.94,E2 -15606.94} C_VEL
LIN {X 0,Y 316.922,Z 532.789,A -85,B 0,C 180,E1 -15608.384,E2 -15608.384} C_VEL
LIN {X 0,Y 316.195,Z 527.521,A -85,B 0,C 180,E1 -15610.913,E2 -15610.913} C_VEL
LIN {X 0,Y 314.943,Z 520.849,A -85,B 0,C 180,E1 -15614.432,E2 -15614.432} C_VEL
LIN {X 0,Y 313.462,Z 513.931,A -85,B 0,C 180,E1 -15618.593,E2 -15618.593} C_VEL
LIN {X 0,Y 312.505,Z 509.556,A -85,B 0,C 180,E1 -15621.633,E2 -15621.633} C_VEL
LIN {X 0,Y 312.534,Z 509.553,A -85,B 0,C 180,E1 -15624.221,E2 -15624.221} C_VEL
LIN {X 0,Y 312.506,Z 509.557,A -85,B 0,C 180,E1 -15627.334,E2 -15627.334} C_VEL
LIN {X 0,Y 312.554,Z 509.547,A -85,B 0,C 180,E1 -15631.277,E2 -15631.277} C_VEL
LIN {X 0,Y 312.588,Z 509.547,A -85,B 0,C 180,E1 -15634.711,E2 -15634.711} C_VEL
LIN {X 0,Y 312.59,Z 509.548,A -85,B 0,C 180,E1 -15637.529,E2 -15637.529} C_VEL
LIN {X 0,Y 312.641,Z 509.536,A -85,B 0,C 180,E1 -15641.657,E2 -15641.657} C_VEL
LIN {X 0,Y 312.697,Z 509.528,A -85,B 0,C 180,E1 -15645.687,E2 -15645.687} C_VEL
LIN {X 0,Y 312.705,Z 509.532,A -85,B 0,C 180,E1 -15649.642,E2 -15649.642} C_VEL
LIN {X 0,Y 312.876,Z 509.505,A -85,B 0,C 180,E1 -15652.255,E2 -15652.255} C_VEL
LIN {X 0,Y 312.713,Z 509.526,A -85,B 0,C 180,E1 -15654.843,E2 -15654.843} C_VEL
LIN {X 0,Y 312.989,Z 509.499,A -85,B 0,C 180,E1 -15658.714,E2 -15658.714} C_VEL
LIN {X 0,Y 312.992,Z 509.499,A -85,B 0,C 180,E1 -15661.287,E2 -15661.287} C_VEL
LIN {X 0,Y 312.707,Z 509.532,A -85,B 0,C 180,E1 -15665.158,E2 -15665.158} C_VEL
LIN {X 0,Y 312.8,Z 509.523,A -85,B 0,C 180,E1 -15667.748,E2 -15667.748} C_VEL
LIN {X 0,Y 312.741,Z 509.527,A -85,B 0,C 180,E1 -15669.491,E2 -15669.491} C_VEL
LIN {X 0,Y 313.001,Z 510.803,A -85,B 0,C 180,E1 -15669.63,E2 -15669.63} C_VEL
LIN {X 0,Y 317.586,Z 520.746,A -85,B 0,C 180,E1 -15671.004,E2 -15671.004} C_VEL
LIN {X 0,Y 321.199,Z 530.366,A -85,B 0,C 180,E1 -15672.398,E2 -15672.398} C_VEL
LIN {X 0,Y 323.8,Z 539.445,A -85,B 0,C 180,E1 -15673.813,E2 -15673.813} C_VEL
LIN {X 0,Y 323.793,Z 541.786,A -85,B 0,C 180,E1 -15674.134,E2 -15674.134} C_VEL
LIN {X 0,Y 322.171,Z 552.417,A -85,B 0,C 180,E1 -15675.65,E2 -15675.65} C_VEL
LIN {X 0,Y 320.633,Z 561.29,A -85,B 0,C 180,E1 -15677.212,E2 -15677.212} C_VEL
LIN {X 0,Y 319.096,Z 569.278,A -85,B 0,C 180,E1 -15678.951,E2 -15678.951} C_VEL
LIN {X 0,Y 317.495,Z 577.074,A -85,B 0,C 180,E1 -15681.109,E2 -15681.109} C_VEL
LIN {X 0,Y 316.325,Z 582.121,A -85,B 0,C 180,E1 -15682.881,E2 -15682.881} C_VEL
LIN {X 0,Y 315.125,Z 586.945,A -85,B 0,C 180,E1 -15685.072,E2 -15685.072} C_VEL
LIN {X 0,Y 314.482,Z 589.467,A -85,B 0,C 180,E1 -15686.63,E2 -15686.63} C_VEL
LIN {X 0,Y 313.633,Z 592.216,A -85,B 0,C 180,E1 -15689.081,E2 -15689.081} C_VEL
LIN {X 0,Y 313.082,Z 593.42,A -85,B 0,C 180,E1 -15691.458,E2 -15691.458} C_VEL
LIN {X 0,Y 312.788,Z 593.316,A -85,B 0,C 180,E1 -15693.762,E2 -15693.762} C_VEL
LIN {X 0,Y 312.726,Z 592.01,A -85,B 0,C 180,E1 -15695.997,E2 -15695.997} C_VEL
LIN {X 0,Y 312.843,Z 589.589,A -85,B 0,C 180,E1 -15698.161,E2 -15698.161} C_VEL
LIN {X 0,Y 313.292,Z 585.392,A -85,B 0,C 180,E1 -15700.584,E2 -15700.584} C_VEL
LIN {X 0,Y 314.003,Z 579.409,A -85,B 0,C 180,E1 -15703.055,E2 -15703.055} C_VEL
LIN {X 0,Y 314.774,Z 572.401,A -85,B 0,C 180,E1 -15705.239,E2 -15705.239} C_VEL
LIN {X 0,Y 315.803,Z 564.216,A -85,B 0,C 180,E1 -15707.257,E2 -15707.257} C_VEL
LIN {X 0,Y 316.767,Z 555.586,A -85,B 0,C 180,E1 -15708.969,E2 -15708.969} C_VEL
LIN {X 0,Y 317.893,Z 544.866,A -85,B 0,C 180,E1 -15710.696,E2 -15710.696} C_VEL
LIN {X 0,Y 318.927,Z 533.824,A -85,B 0,C 180,E1 -15712.116,E2 -15712.116} C_VEL
LIN {X 0,Y 318.577,Z 530.591,A -85,B 0,C 180,E1 -15712.516,E2 -15712.516} C_VEL
LIN {X 0,Y 315.294,Z 518.749,A -85,B 0,C 180,E1 -15713.896,E2 -15713.896} C_VEL
LIN {X 0,Y 312.53,Z 509.554,A -85,B 0,C 180,E1 -15714.813,E2 -15714.813} C_VEL
LIN {X 0,Y 312.528,Z 509.554,A -85,B 0,C 180,E1 -15718.854,E2 -15718.854} C_VEL
LIN {X 0,Y 312.579,Z 509.548,A -85,B 0,C 180,E1 -15721.825,E2 -15721.825} C_VEL
LIN {X 0,Y 312.59,Z 509.545,A -85,B 0,C 180,E1 -15724.711,E2 -15724.711} C_VEL
LIN {X 0,Y 312.569,Z 509.551,A -85,B 0,C 180,E1 -15727.527,E2 -15727.527} C_VEL
LIN {X 0,Y 312.587,Z 509.548,A -85,B 0,C 180,E1 -15731.653,E2 -15731.653} C_VEL
LIN {X 0,Y 312.69,Z 509.534,A -85,B 0,C 180,E1 -15735.686,E2 -15735.686} C_VEL
LIN {X 0,Y 312.691,Z 509.535,A -85,B 0,C 180,E1 -15739.641,E2 -15739.641} C_VEL
LIN {X 0,Y 312.801,Z 509.518,A -85,B 0,C 180,E1 -15742.252,E2 -15742.252} C_VEL
LIN {X 0,Y 312.708,Z 509.531,A -85,B 0,C 180,E1 -15744.842,E2 -15744.842} C_VEL
LIN {X 0,Y 312.94,Z 509.505,A -85,B 0,C 180,E1 -15747.425,E2 -15747.425} C_VEL
LIN {X 0,Y 313.043,Z 509.488,A -85,B 0,C 180,E1 -15750,E2 -15750} C_VEL
LIN {X 0,Y 312.936,Z 509.502,A -85,B 0,C 180,E1 -15752.574,E2 -15752.574} C_VEL
LIN {X 0,Y 312.848,Z 509.512,A -85,B 0,C 180,E1 -15756.449,E2 -15756.449} C_VEL
LIN {X 0,Y 312.755,Z 509.527,A -85,B 0,C 180,E1 -15759.05,E2 -15759.05} C_VEL
LIN {X 0,Y 312.639,Z 509.542,A -85,B 0,C 180,E1 -15762.991,E2 -15762.991} C_VEL
LIN {X 0,Y 312.626,Z 509.541,A -85,B 0,C 180,E1 -15765.65,E2 -15765.65} C_VEL
LIN {X 0,Y 312.583,Z 509.547,A -85,B 0,C 180,E1 -15769.71,E2 -15769.71} C_VEL
LIN {X 0,Y 312.549,Z 509.551,A -85,B 0,C 180,E1 -15772.789,E2 -15772.789} C_VEL
LIN {X 0,Y 312.542,Z 509.55,A -85,B 0,C 180,E1 -15775.911,E2 -15775.911} C_VEL
LIN {X 0,Y 312.507,Z 509.556,A -85,B 0,C 180,E1 -15779.654,E2 -15779.654} C_VEL
LIN {X 0,Y 312.523,Z 509.553,A -85,B 0,C 180,E1 -15783.688,E2 -15783.688} C_VEL
LIN {X 0,Y 312.517,Z 509.557,A -85,B 0,C 180,E1 -15787.386,E2 -15787.386} C_VEL
LIN {X 0,Y 312.444,Z 509.565,A -85,B 0,C 180,E1 -15790.717,E2 -15790.717} C_VEL
LIN {X 0,Y 312.454,Z 509.561,A -85,B 0,C 180,E1 -15794.209,E2 -15794.209} C_VEL
LIN {X 0,Y 312.487,Z 509.557,A -85,B 0,C 180,E1 -15797.918,E2 -15797.918} C_VEL
LIN {X 0,Y 312.501,Z 509.56,A -85,B 0,C 180,E1 -15800.971,E2 -15800.971} C_VEL
LIN {X 0,Y 312.534,Z 509.551,A -85,B 0,C 180,E1 -15804.22,E2 -15804.22} C_VEL
LIN {X 0,Y 312.507,Z 509.558,A -85,B 0,C 180,E1 -15807.334,E2 -15807.334} C_VEL
LIN {X 0,Y 312.555,Z 509.552,A -85,B 0,C 180,E1 -15811.276,E2 -15811.276} C_VEL
LIN {X 0,Y 312.587,Z 509.547,A -85,B 0,C 180,E1 -15814.711,E2 -15814.711} C_VEL
LIN {X 0,Y 312.539,Z 509.555,A -85,B 0,C 180,E1 -15818.912,E2 -15818.912} C_VEL
LIN {X 0,Y 312.641,Z 509.539,A -85,B 0,C 180,E1 -15821.656,E2 -15821.656} C_VEL
LIN {X 0,Y 312.696,Z 509.531,A -85,B 0,C 180,E1 -15825.686,E2 -15825.686} C_VEL
LIN {X 0,Y 312.687,Z 509.533,A -85,B 0,C 180,E1 -15829.688,E2 -15829.688} C_VEL
LIN {X 0,Y 312.024,Z 509.619,A -85,B 0,C 180,E1 -15830.765,E2 -15830.765} C_VEL
LIN {X 0,Y 309.183,Z 509.971,A -85,B 0,C 180,E1 -15832.519,E2 -15832.519} C_VEL
LIN {X 0,Y 306.768,Z 510.271,A -85,B 0,C 180,E1 -15833.941,E2 -15833.941} C_VEL
LIN {X 0,Y 305.724,Z 510.404,A -85,B 0,C 180,E1 -15835.042,E2 -15835.042} C_VEL
LIN {X 0,Y 305.634,Z 510.41,A -85,B 0,C 180,E1 -15835.415,E2 -15835.415} C_VEL
LIN {X 0,Y 305.954,Z 510.374,A -85,B 0,C 180,E1 -15838.683,E2 -15838.683} C_VEL
LIN {X 0,Y 305.955,Z 510.373,A -85,B 0,C 180,E1 -15841.316,E2 -15841.316} C_VEL
LIN {X 0,Y 305.665,Z 510.409,A -85,B 0,C 180,E1 -15845.277,E2 -15845.277} C_VEL
LIN {X 0,Y 305.748,Z 510.397,A -85,B 0,C 180,E1 -15847.927,E2 -15847.927} C_VEL
LIN {X 0,Y 305.607,Z 510.414,A -85,B 0,C 180,E1 -15851.945,E2 -15851.945} C_VEL
LIN {X 0,Y 305.61,Z 510.418,A -85,B 0,C 180,E1 -15855.014,E2 -15855.014} C_VEL
LIN {X 0,Y 305.543,Z 510.423,A -85,B 0,C 180,E1 -15859.426,E2 -15859.426} C_VEL
LIN {X 0,Y 305.487,Z 510.433,A -85,B 0,C 180,E1 -15863.039,E2 -15863.039} C_VEL
LIN {X 0,Y 305.474,Z 510.432,A -85,B 0,C 180,E1 -15866.199,E2 -15866.199} C_VEL
LIN {X 0,Y 305.459,Z 510.436,A -85,B 0,C 180,E1 -15869.037,E2 -15869.037} C_VEL
LIN {X 0,Y 305.437,Z 510.436,A -85,B 0,C 180,E1 -15871.953,E2 -15871.953} C_VEL
LIN {X 0,Y 305.463,Z 510.435,A -85,B 0,C 180,E1 -15875.113,E2 -15875.113} C_VEL
LIN {X 0,Y 305.45,Z 510.438,A -85,B 0,C 180,E1 -15878.529,E2 -15878.529} C_VEL
LIN {X 0,Y 305.486,Z 510.455,A -85,B 0,C 180,E1 -15881.164,E2 -15881.164} C_VEL
LIN {X 0,Y 307.103,Z 518.795,A -85,B 0,C 180,E1 -15885.188,E2 -15885.188} C_VEL
LIN {X 0,Y 308.791,Z 527.545,A -85,B 0,C 180,E1 -15889.167,E2 -15889.167} C_VEL
LIN {X 0,Y 309.763,Z 532.706,A -85,B 0,C 180,E1 -15891.418,E2 -15891.418} C_VEL
LIN {X 0,Y 309.697,Z 535.546,A -85,B 0,C 180,E1 -15892.585,E2 -15892.585} C_VEL
LIN {X 0,Y 308.148,Z 546.179,A -85,B 0,C 180,E1 -15896.813,E2 -15896.813} C_VEL
LIN {X 0,Y 306.652,Z 557.513,A -85,B 0,C 180,E1 -15901.23,E2 -15901.23} C_VEL
LIN {X 0,Y 305.558,Z 568.748,A -85,B 0,C 180,E1 -15905.543,E2 -15905.543} C_VEL
LIN {X 0,Y 305.133,Z 573.613,A -85,B 0,C 180,E1 -15907.396,E2 -15907.396} C_VEL
LIN {X 0,Y 306.768,Z 589.838,A -85,B 0,C 180,E1 -15908.232,E2 -15908.232} C_VEL
LIN {X 0,Y 307.708,Z 602.704,A -85,B 0,C 180,E1 -15909.15,E2 -15909.15} C_VEL
LIN {X 0,Y 308.202,Z 615.736,A -85,B 0,C 180,E1 -15910.346,E2 -15910.346} C_VEL
LIN {X 0,Y 308.341,Z 627.667,A -85,B 0,C 180,E1 -15911.736,E2 -15911.736} C_VEL
LIN {X 0,Y 307.965,Z 633.816,A -85,B 0,C 180,E1 -15912.571,E2 -15912.571} C_VEL
LIN {X 0,Y 306.743,Z 644.112,A -85,B 0,C 180,E1 -15914.215,E2 -15914.215} C_VEL
LIN {X 0,Y 305.653,Z 653.209,A -85,B 0,C 180,E1 -15916.029,E2 -15916.029} C_VEL
LIN {X 0,Y 304.971,Z 661.318,A -85,B 0,C 180,E1 -15918.03,E2 -15918.03} C_VEL
LIN {X 0,Y 304.622,Z 667.828,A -85,B 0,C 180,E1 -15920.036,E2 -15920.036} C_VEL
LIN {X 0,Y 304.559,Z 672.964,A -85,B 0,C 180,E1 -15922.042,E2 -15922.042} C_VEL
LIN {X 0,Y 304.718,Z 676.905,A -85,B 0,C 180,E1 -15924.043,E2 -15924.043} C_VEL
LIN {X 0,Y 304.967,Z 679.74,A -85,B 0,C 180,E1 -15926.036,E2 -15926.036} C_VEL
LIN {X 0,Y 305.089,Z 681.017,A -85,B 0,C 180,E1 -15927.36,E2 -15927.36} C_VEL
LIN {X 0,Y 305.277,Z 681.873,A -85,B 0,C 180,E1 -15928.681,E2 -15928.681} C_VEL
LIN {X 0,Y 305.499,Z 682.313,A -85,B 0,C 180,E1 -15930,E2 -15930} C_VEL
LIN {X 0,Y 305.158,Z 682.211,A -85,B 0,C 180,E1 -15931.32,E2 -15931.32} C_VEL
LIN {X 0,Y 305.006,Z 681.694,A -85,B 0,C 180,E1 -15932.642,E2 -15932.642} C_VEL
LIN {X 0,Y 304.909,Z 680.773,A -85,B 0,C 180,E1 -15933.965,E2 -15933.965} C_VEL
LIN {X 0,Y 304.669,Z 679.414,A -85,B 0,C 180,E1 -15935.294,E2 -15935.294} C_VEL
LIN {X 0,Y 304.481,Z 676.994,A -85,B 0,C 180,E1 -15937.012,E2 -15937.012} C_VEL
LIN {X 0,Y 304.39,Z 672.641,A -85,B 0,C 180,E1 -15939.301,E2 -15939.301} C_VEL
LIN {X 0,Y 304.631,Z 667.666,A -85,B 0,C 180,E1 -15941.309,E2 -15941.309} C_VEL
LIN {X 0,Y 305.426,Z 660.358,A -85,B 0,C 180,E1 -15943.642,E2 -15943.642} C_VEL
LIN {X 0,Y 306.541,Z 652.167,A -85,B 0,C 180,E1 -15945.728,E2 -15945.728} C_VEL
LIN {X 0,Y 308.176,Z 643.144,A -85,B 0,C 180,E1 -15947.588,E2 -15947.588} C_VEL
LIN {X 0,Y 309.92,Z 633.592,A -85,B 0,C 180,E1 -15949.197,E2 -15949.197} C_VEL
LIN {X 0,Y 310.639,Z 623.161,A -85,B 0,C 180,E1 -15950.702,E2 -15950.702} C_VEL
LIN {X 0,Y 311.362,Z 610.041,A -85,B 0,C 180,E1 -15952.264,E2 -15952.264} C_VEL
LIN {X 0,Y 311.106,Z 597.676,A -85,B 0,C 180,E1 -15953.512,E2 -15953.512} C_VEL
LIN {X 0,Y 309.761,Z 584.869,A -85,B 0,C 180,E1 -15954.639,E2 -15954.639} C_VEL
LIN {X 0,Y 307.22,Z 570.961,A -85,B 0,C 180,E1 -15955.727,E2 -15955.727} C_VEL
LIN {X 0,Y 305.912,Z 564.437,A -85,B 0,C 180,E1 -15956.179,E2 -15956.179} C_VEL
LIN {X 0,Y 307.018,Z 554.003,A -85,B 0,C 180,E1 -15960.239,E2 -15960.239} C_VEL
LIN {X 0,Y 308.59,Z 543,A -85,B 0,C 180,E1 -15964.706,E2 -15964.706} C_VEL
LIN {X 0,Y 309.902,Z 535.825,A -85,B 0,C 180,E1 -15967.757,E2 -15967.757} C_VEL
LIN {X 0,Y 309.803,Z 532.038,A -85,B 0,C 180,E1 -15969.529,E2 -15969.529} C_VEL
LIN {X 0,Y 308.51,Z 524.977,A -85,B 0,C 180,E1 -15973.2,E2 -15973.2} C_VEL
LIN {X 0,Y 307.287,Z 519.01,A -85,B 0,C 180,E1 -15976.675,E2 -15976.675} C_VEL
LIN {X 0,Y 306.198,Z 513.945,A -85,B 0,C 180,E1 -15980.009,E2 -15980.009} C_VEL
LIN {X 0,Y 305.484,Z 510.434,A -85,B 0,C 180,E1 -15982.643,E2 -15982.643} C_VEL
LIN {X 0,Y 305.467,Z 510.432,A -85,B 0,C 180,E1 -15986.484,E2 -15986.484} C_VEL
LIN {X 0,Y 305.498,Z 510.424,A -85,B 0,C 180,E1 -15990.95,E2 -15990.95} C_VEL
LIN {X 0,Y 305.574,Z 510.417,A -85,B 0,C 180,E1 -15994.088,E2 -15994.088} C_VEL
LIN {X 0,Y 305.503,Z 510.425,A -85,B 0,C 180,E1 -15998.403,E2 -15998.403} C_VEL
LIN {X 0,Y 305.593,Z 510.417,A -85,B 0,C 180,E1 -16001.218,E2 -16001.218} C_VEL
LIN {X 0,Y 305.652,Z 510.405,A -85,B 0,C 180,E1 -16005.349,E2 -16005.349} C_VEL
LIN {X 0,Y 305.642,Z 510.41,A -85,B 0,C 180,E1 -16009.4,E2 -16009.4} C_VEL
LIN {X 0,Y 305.816,Z 510.384,A -85,B 0,C 180,E1 -16012.075,E2 -16012.075} C_VEL
LIN {X 0,Y 305.685,Z 510.402,A -85,B 0,C 180,E1 -16014.724,E2 -16014.724} C_VEL
LIN {X 0,Y 305.956,Z 510.375,A -85,B 0,C 180,E1 -16018.684,E2 -16018.684} C_VEL
LIN {X 0,Y 305.959,Z 510.375,A -85,B 0,C 180,E1 -16021.317,E2 -16021.317} C_VEL
LIN {X 0,Y 305.675,Z 510.406,A -85,B 0,C 180,E1 -16025.277,E2 -16025.277} C_VEL
LIN {X 0,Y 305.784,Z 510.391,A -85,B 0,C 180,E1 -16028.595,E2 -16028.595} C_VEL
LIN {X 0,Y 305.871,Z 510.98,A -85,B 0,C 180,E1 -16028.703,E2 -16028.703} C_VEL
LIN {X 0,Y 306.778,Z 513.327,A -85,B 0,C 180,E1 -16029.008,E2 -16029.008} C_VEL
LIN {X 0,Y 311.218,Z 522.901,A -85,B 0,C 180,E1 -16030.408,E2 -16030.408} C_VEL
LIN {X 0,Y 314.623,Z 531.921,A -85,B 0,C 180,E1 -16031.799,E2 -16031.799} C_VEL
LIN {X 0,Y 317.492,Z 541.984,A -85,B 0,C 180,E1 -16033.44,E2 -16033.44} C_VEL
LIN {X 0,Y 316.151,Z 551.617,A -85,B 0,C 180,E1 -16034.812,E2 -16034.812} C_VEL
LIN {X 0,Y 314.435,Z 561.008,A -85,B 0,C 180,E1 -16036.444,E2 -16036.444} C_VEL
LIN {X 0,Y 312.668,Z 569.773,A -85,B 0,C 180,E1 -16038.342,E2 -16038.342} C_VEL
LIN {X 0,Y 311.253,Z 576.397,A -85,B 0,C 180,E1 -16040.142,E2 -16040.142} C_VEL
LIN {X 0,Y 309.837,Z 582.221,A -85,B 0,C 180,E1 -16042.114,E2 -16042.114} C_VEL
LIN {X 0,Y 308.543,Z 587.248,A -85,B 0,C 180,E1 -16044.338,E2 -16044.338} C_VEL
LIN {X 0,Y 307.896,Z 589.649,A -85,B 0,C 180,E1 -16045.703,E2 -16045.703} C_VEL
LIN {X 0,Y 307.27,Z 591.698,A -85,B 0,C 180,E1 -16047.223,E2 -16047.223} C_VEL
LIN {X 0,Y 306.529,Z 593.678,A -85,B 0,C 180,E1 -16049.395,E2 -16049.395} C_VEL
LIN {X 0,Y 305.995,Z 594.609,A -85,B 0,C 180,E1 -16051.888,E2 -16051.888} C_VEL
LIN {X 0,Y 305.749,Z 594.197,A -85,B 0,C 180,E1 -16054.156,E2 -16054.156} C_VEL
LIN {X 0,Y 305.72,Z 592.325,A -85,B 0,C 180,E1 -16056.706,E2 -16056.706} C_VEL
LIN {X 0,Y 305.959,Z 588.945,A -85,B 0,C 180,E1 -16059.257,E2 -16059.257} C_VEL
LIN {X 0,Y 306.537,Z 584.145,A -85,B 0,C 180,E1 -16061.674,E2 -16061.674} C_VEL
LIN {X 0,Y 307.197,Z 578.697,A -85,B 0,C 180,E1 -16063.75,E2 -16063.75} C_VEL
LIN {X 0,Y 307.839,Z 572.932,A -85,B 0,C 180,E1 -16065.517,E2 -16065.517} C_VEL
LIN {X 0,Y 308.731,Z 566.113,A -85,B 0,C 180,E1 -16067.235,E2 -16067.235} C_VEL
LIN {X 0,Y 309.803,Z 556.967,A -85,B 0,C 180,E1 -16069.122,E2 -16069.122} C_VEL
LIN {X 0,Y 310.986,Z 545.99,A -85,B 0,C 180,E1 -16070.936,E2 -16070.936} C_VEL
LIN {X 0,Y 312.039,Z 534.995,A -85,B 0,C 180,E1 -16072.386,E2 -16072.386} C_VEL
LIN {X 0,Y 311.828,Z 532.536,A -85,B 0,C 180,E1 -16072.695,E2 -16072.695} C_VEL
LIN {X 0,Y 308.664,Z 521.012,A -85,B 0,C 180,E1 -16074.104,E2 -16074.104} C_VEL
LIN {X 0,Y 305.486,Z 510.434,A -85,B 0,C 180,E1 -16075.214,E2 -16075.214} C_VEL
LIN {X 0,Y 305.468,Z 510.436,A -85,B 0,C 180,E1 -16079.591,E2 -16079.591} C_VEL
LIN {X 0,Y 305.539,Z 510.424,A -85,B 0,C 180,E1 -16082.61,E2 -16082.61} C_VEL
LIN {X 0,Y 305.51,Z 510.431,A -85,B 0,C 180,E1 -16085.539,E2 -16085.539} C_VEL
LIN {X 0,Y 305.501,Z 510.429,A -85,B 0,C 180,E1 -16089.813,E2 -16089.813} C_VEL
LIN {X 0,Y 305.547,Z 510.422,A -85,B 0,C 180,E1 -16092.601,E2 -16092.601} C_VEL
LIN {X 0,Y 305.631,Z 510.417,A -85,B 0,C 180,E1 -16095.348,E2 -16095.348} C_VEL
LIN {X 0,Y 305.63,Z 510.416,A -85,B 0,C 180,E1 -16099.399,E2 -16099.399} C_VEL
LIN {X 0,Y 305.751,Z 510.397,A -85,B 0,C 180,E1 -16102.073,E2 -16102.073} C_VEL
LIN {X 0,Y 305.677,Z 510.407,A -85,B 0,C 180,E1 -16104.723,E2 -16104.723} C_VEL
LIN {X 0,Y 305.955,Z 510.372,A -85,B 0,C 180,E1 -16108.684,E2 -16108.684} C_VEL
LIN {X 0,Y 305.958,Z 510.376,A -85,B 0,C 180,E1 -16111.316,E2 -16111.316} C_VEL
LIN {X 0,Y 305.672,Z 510.412,A -85,B 0,C 180,E1 -16115.277,E2 -16115.277} C_VEL
LIN {X 0,Y 305.751,Z 510.396,A -85,B 0,C 180,E1 -16117.927,E2 -16117.927} C_VEL
LIN {X 0,Y 305.604,Z 510.415,A -85,B 0,C 180,E1 -16121.945,E2 -16121.945} C_VEL
LIN {X 0,Y 305.613,Z 510.417,A -85,B 0,C 180,E1 -16125.015,E2 -16125.015} C_VEL
LIN {X 0,Y 305.565,Z 510.423,A -85,B 0,C 180,E1 -16129.436,E2 -16129.436} C_VEL
LIN {X 0,Y 305.492,Z 510.433,A -85,B 0,C 180,E1 -16133.04,E2 -16133.04} C_VEL
LIN {X 0,Y 305.481,Z 510.429,A -85,B 0,C 180,E1 -16136.2,E2 -16136.2} C_VEL
LIN {X 0,Y 305.467,Z 510.436,A -85,B 0,C 180,E1 -16139.039,E2 -16139.039} C_VEL
LIN {X 0,Y 305.44,Z 510.435,A -85,B 0,C 180,E1 -16141.953,E2 -16141.953} C_VEL
LIN {X 0,Y 305.465,Z 510.437,A -85,B 0,C 180,E1 -16145.113,E2 -16145.113} C_VEL
LIN {X 0,Y 305.436,Z 510.436,A -85,B 0,C 180,E1 -16148.524,E2 -16148.524} C_VEL
LIN {X 0,Y 305.438,Z 510.436,A -85,B 0,C 180,E1 -16152.581,E2 -16152.581} C_VEL
LIN {X 0,Y 305.428,Z 510.437,A -85,B 0,C 180,E1 -16156.345,E2 -16156.345} C_VEL
LIN {X 0,Y 305.46,Z 510.432,A -85,B 0,C 180,E1 -16159.892,E2 -16159.892} C_VEL
LIN {X 0,Y 305.483,Z 510.431,A -85,B 0,C 180,E1 -16163.631,E2 -16163.631} C_VEL
LIN {X 0,Y 305.468,Z 510.433,A -85,B 0,C 180,E1 -16166.483,E2 -16166.483} C_VEL
LIN {X 0,Y 305.499,Z 510.432,A -85,B 0,C 180,E1 -16170.95,E2 -16170.95} C_VEL
LIN {X 0,Y 305.574,Z 510.418,A -85,B 0,C 180,E1 -16174.088,E2 -16174.088} C_VEL
LIN {X 0,Y 305.483,Z 510.43,A -85,B 0,C 180,E1 -16178.401,E2 -16178.401} C_VEL
LIN {X 0,Y 305.592,Z 510.419,A -85,B 0,C 180,E1 -16181.217,E2 -16181.217} C_VEL
LIN {X 0,Y 305.651,Z 510.411,A -85,B 0,C 180,E1 -16185.349,E2 -16185.349} C_VEL
LIN {X 0,Y 305.627,Z 510.412,A -85,B 0,C 180,E1 -16189.692,E2 -16189.692} C_VEL
LIN {X 0,Y 305.753,Z 510.396,A -85,B 0,C 180,E1 -16192.072,E2 -16192.072} C_VEL
LIN {X 0,Y 305.674,Z 510.409,A -85,B 0,C 180,E1 -16194.723,E2 -16194.723} C_VEL
LIN {X 0,Y 305.634,Z 510.41,A -85,B 0,C 180,E1 -16195.415,E2 -16195.415} C_VEL
LIN {X 0,Y 304.986,Z 510.495,A -85,B 0,C 180,E1 -16196.517,E2 -16196.517} C_VEL
LIN {X 0,Y 302.26,Z 510.832,A -85,B 0,C 180,E1 -16198.315,E2 -16198.315} C_VEL
LIN {X 0,Y 299.966,Z 511.117,A -85,B 0,C 180,E1 -16199.774,E2 -16199.774} C_VEL
LIN {X 0,Y 298.994,Z 511.244,A -85,B 0,C 180,E1 -16200.9,E2 -16200.9} C_VEL
LIN {X 0,Y 298.92,Z 511.248,A -85,B 0,C 180,E1 -16201.281,E2 -16201.281} C_VEL
LIN {X 0,Y 298.634,Z 511.284,A -85,B 0,C 180,E1 -16205.401,E2 -16205.401} C_VEL
LIN {X 0,Y 298.699,Z 511.275,A -85,B 0,C 180,E1 -16208.115,E2 -16208.115} C_VEL
LIN {X 0,Y 298.557,Z 511.293,A -85,B 0,C 180,E1 -16212.231,E2 -16212.231} C_VEL
LIN {X 0,Y 298.549,Z 511.296,A -85,B 0,C 180,E1 -16215.168,E2 -16215.168} C_VEL
LIN {X 0,Y 298.504,Z 511.301,A -85,B 0,C 180,E1 -16219.245,E2 -16219.245} C_VEL
LIN {X 0,Y 298.424,Z 511.309,A -85,B 0,C 180,E1 -16223.6,E2 -16223.6} C_VEL
LIN {X 0,Y 298.413,Z 511.314,A -85,B 0,C 180,E1 -16226.582,E2 -16226.582} C_VEL
LIN {X 0,Y 298.398,Z 511.312,A -85,B 0,C 180,E1 -16229.643,E2 -16229.643} C_VEL
LIN {X 0,Y 298.393,Z 511.319,A -85,B 0,C 180,E1 -16232.8,E2 -16232.8} C_VEL
LIN {X 0,Y 298.447,Z 511.311,A -85,B 0,C 180,E1 -16236.807,E2 -16236.807} C_VEL
LIN {X 0,Y 298.451,Z 511.456,A -85,B 0,C 180,E1 -16240.852,E2 -16240.852} C_VEL
LIN {X 0,Y 299.959,Z 519.166,A -85,B 0,C 180,E1 -16244.66,E2 -16244.66} C_VEL
LIN {X 0,Y 301.426,Z 526.815,A -85,B 0,C 180,E1 -16248.254,E2 -16248.254} C_VEL
LIN {X 0,Y 302.692,Z 533.312,A -85,B 0,C 180,E1 -16251.179,E2 -16251.179} C_VEL
LIN {X 0,Y 302.809,Z 535.475,A -85,B 0,C 180,E1 -16252.103,E2 -16252.103} C_VEL
LIN {X 0,Y 301.116,Z 546.625,A -85,B 0,C 180,E1 -16256.657,E2 -16256.657} C_VEL
LIN {X 0,Y 299.539,Z 558.148,A -85,B 0,C 180,E1 -16261.25,E2 -16261.25} C_VEL
LIN {X 0,Y 298.442,Z 569.292,A -85,B 0,C 180,E1 -16265.663,E2 -16265.663} C_VEL
LIN {X 0,Y 298.131,Z 572.681,A -85,B 0,C 180,E1 -16266.993,E2 -16266.993} C_VEL
LIN {X 0,Y 299.663,Z 588.452,A -85,B 0,C 180,E1 -16267.813,E2 -16267.813} C_VEL
LIN {X 0,Y 300.597,Z 601.433,A -85,B 0,C 180,E1 -16268.757,E2 -16268.757} C_VEL
LIN {X 0,Y 301.127,Z 613.362,A -85,B 0,C 180,E1 -16269.864,E2 -16269.864} C_VEL
LIN {X 0,Y 301.303,Z 624.304,A -85,B 0,C 180,E1 -16271.117,E2 -16271.117} C_VEL
LIN {X 0,Y 301.205,Z 632.006,A -85,B 0,C 180,E1 -16272.167,E2 -16272.167} C_VEL
LIN {X 0,Y 299.99,Z 641.461,A -85,B 0,C 180,E1 -16273.672,E2 -16273.672} C_VEL
LIN {X 0,Y 298.845,Z 650.126,A -85,B 0,C 180,E1 -16275.356,E2 -16275.356} C_VEL
LIN {X 0,Y 298.192,Z 657.349,A -85,B 0,C 180,E1 -16277.062,E2 -16277.062} C_VEL
LIN {X 0,Y 297.664,Z 664.42,A -85,B 0,C 180,E1 -16279.112,E2 -16279.112} C_VEL
LIN {X 0,Y 297.504,Z 670.062,A -85,B 0,C 180,E1 -16281.167,E2 -16281.167} C_VEL
LIN {X 0,Y 297.567,Z 674.452,A -85,B 0,C 180,E1 -16283.218,E2 -16283.218} C_VEL
LIN {X 0,Y 297.778,Z 676.753,A -85,B 0,C 180,E1 -16284.583,E2 -16284.583} C_VEL
LIN {X 0,Y 297.921,Z 678.573,A -85,B 0,C 180,E1 -16285.942,E2 -16285.942} C_VEL
LIN {X 0,Y 298.052,Z 679.885,A -85,B 0,C 180,E1 -16287.297,E2 -16287.297} C_VEL
LIN {X 0,Y 298.265,Z 680.769,A -85,B 0,C 180,E1 -16288.65,E2 -16288.65} C_VEL
LIN {X 0,Y 298.489,Z 681.231,A -85,B 0,C 180,E1 -16290,E2 -16290} C_VEL
LIN {X 0,Y 298.121,Z 681.172,A -85,B 0,C 180,E1 -16291.351,E2 -16291.351} C_VEL
LIN {X 0,Y 297.959,Z 680.682,A -85,B 0,C 180,E1 -16292.704,E2 -16292.704} C_VEL
LIN {X 0,Y 297.855,Z 679.783,A -85,B 0,C 180,E1 -16294.059,E2 -16294.059} C_VEL
LIN {X 0,Y 297.582,Z 678.44,A -85,B 0,C 180,E1 -16295.421,E2 -16295.421} C_VEL
LIN {X 0,Y 297.402,Z 676.326,A -85,B 0,C 180,E1 -16297.015,E2 -16297.015} C_VEL
LIN {X 0,Y 297.307,Z 671.759,A -85,B 0,C 180,E1 -16299.525,E2 -16299.525} C_VEL
LIN {X 0,Y 297.611,Z 666.868,A -85,B 0,C 180,E1 -16301.58,E2 -16301.58} C_VEL
LIN {X 0,Y 298.481,Z 659.695,A -85,B 0,C 180,E1 -16303.966,E2 -16303.966} C_VEL
LIN {X 0,Y 299.459,Z 652.632,A -85,B 0,C 180,E1 -16305.855,E2 -16305.855} C_VEL
LIN {X 0,Y 301.069,Z 644.365,A -85,B 0,C 180,E1 -16307.666,E2 -16307.666} C_VEL
LIN {X 0,Y 303.016,Z 634.271,A -85,B 0,C 180,E1 -16309.476,E2 -16309.476} C_VEL
LIN {X 0,Y 303.937,Z 623.155,A -85,B 0,C 180,E1 -16311.18,E2 -16311.18} C_VEL
LIN {X 0,Y 304.736,Z 610.942,A -85,B 0,C 180,E1 -16312.705,E2 -16312.705} C_VEL
LIN {X 0,Y 304.572,Z 597.967,A -85,B 0,C 180,E1 -16314.091,E2 -16314.091} C_VEL
LIN {X 0,Y 303.251,Z 584.752,A -85,B 0,C 180,E1 -16315.332,E2 -16315.332} C_VEL
LIN {X 0,Y 300.756,Z 570.699,A -85,B 0,C 180,E1 -16316.501,E2 -16316.501} C_VEL
LIN {X 0,Y 299.044,Z 562.982,A -85,B 0,C 180,E1 -16317.106,E2 -16317.106} C_VEL
LIN {X 0,Y 300.195,Z 553.307,A -85,B 0,C 180,E1 -16321.001,E2 -16321.001} C_VEL
LIN {X 0,Y 301.861,Z 542.785,A -85,B 0,C 180,E1 -16325.425,E2 -16325.425} C_VEL
LIN {X 0,Y 302.995,Z 537.033,A -85,B 0,C 180,E1 -16327.942,E2 -16327.942} C_VEL
LIN {X 0,Y 302.946,Z 534.049,A -85,B 0,C 180,E1 -16329.373,E2 -16329.373} C_VEL
LIN {X 0,Y 301.685,Z 527.039,A -85,B 0,C 180,E1 -16333.093,E2 -16333.093} C_VEL
LIN {X 0,Y 300.558,Z 521.367,A -85,B 0,C 180,E1 -16336.459,E2 -16336.459} C_VEL
LIN {X 0,Y 299.499,Z 516.325,A -85,B 0,C 180,E1 -16339.811,E2 -16339.811} C_VEL
LIN {X 0,Y 298.433,Z 511.308,A -85,B 0,C 180,E1 -16343.689,E2 -16343.689} C_VEL
LIN {X 0,Y 298.398,Z 511.316,A -85,B 0,C 180,E1 -16347.2,E2 -16347.2} C_VEL
LIN {X 0,Y 298.434,Z 511.304,A -85,B 0,C 180,E1 -16350.615,E2 -16350.615} C_VEL
LIN {X 0,Y 298.486,Z 511.296,A -85,B 0,C 180,E1 -16353.474,E2 -16353.474} C_VEL
LIN {X 0,Y 298.438,Z 511.304,A -85,B 0,C 180,E1 -16356.698,E2 -16356.698} C_VEL
LIN {X 0,Y 298.542,Z 511.298,A -85,B 0,C 180,E1 -16360.757,E2 -16360.757} C_VEL
LIN {X 0,Y 298.596,Z 511.284,A -85,B 0,C 180,E1 -16364.995,E2 -16364.995} C_VEL
LIN {X 0,Y 298.597,Z 511.285,A -85,B 0,C 180,E1 -16369.147,E2 -16369.147} C_VEL
LIN {X 0,Y 298.762,Z 511.262,A -85,B 0,C 180,E1 -16371.886,E2 -16371.886} C_VEL
LIN {X 0,Y 298.657,Z 511.278,A -85,B 0,C 180,E1 -16374.599,E2 -16374.599} C_VEL
LIN {X 0,Y 298.922,Z 511.251,A -85,B 0,C 180,E1 -16378.653,E2 -16378.653} C_VEL
LIN {X 0,Y 298.926,Z 511.251,A -85,B 0,C 180,E1 -16381.348,E2 -16381.348} C_VEL
LIN {X 0,Y 298.643,Z 511.281,A -85,B 0,C 180,E1 -16385.402,E2 -16385.402} C_VEL
LIN {X 0,Y 298.721,Z 511.277,A -85,B 0,C 180,E1 -16387.69,E2 -16387.69} C_VEL
LIN {X 0,Y 299.788,Z 514.235,A -85,B 0,C 180,E1 -16388.086,E2 -16388.086} C_VEL
LIN {X 0,Y 300.453,Z 515.088,A -85,B 0,C 180,E1 -16388.251,E2 -16388.251} C_VEL
LIN {X 0,Y 305.459,Z 526.402,A -85,B 0,C 180,E1 -16390,E2 -16390} C_VEL
LIN {X 0,Y 308.754,Z 535.53,A -85,B 0,C 180,E1 -16391.489,E2 -16391.489} C_VEL
LIN {X 0,Y 311.16,Z 544.5,A -85,B 0,C 180,E1 -16393.054,E2 -16393.054} C_VEL
LIN {X 0,Y 309.406,Z 555.07,A -85,B 0,C 180,E1 -16394.638,E2 -16394.638} C_VEL
LIN {X 0,Y 307.613,Z 564.273,A -85,B 0,C 180,E1 -16396.346,E2 -16396.346} C_VEL
LIN {X 0,Y 305.659,Z 573.117,A -85,B 0,C 180,E1 -16398.431,E2 -16398.431} C_VEL
LIN {X 0,Y 304.194,Z 579.342,A -85,B 0,C 180,E1 -16400.277,E2 -16400.277} C_VEL
LIN {X 0,Y 302.615,Z 585.332,A -85,B 0,C 180,E1 -16402.532,E2 -16402.532} C_VEL
LIN {X 0,Y 301.272,Z 589.849,A -85,B 0,C 180,E1 -16404.829,E2 -16404.829} C_VEL
LIN {X 0,Y 300.278,Z 593.092,A -85,B 0,C 180,E1 -16407.202,E2 -16407.202} C_VEL
LIN {X 0,Y 299.46,Z 595.104,A -85,B 0,C 180,E1 -16409.732,E2 -16409.732} C_VEL
LIN {X 0,Y 298.94,Z 595.675,A -85,B 0,C 180,E1 -16412.182,E2 -16412.182} C_VEL
LIN {X 0,Y 298.715,Z 594.988,A -85,B 0,C 180,E1 -16414.567,E2 -16414.567} C_VEL
LIN {X 0,Y 298.691,Z 593.156,A -85,B 0,C 180,E1 -16416.869,E2 -16416.869} C_VEL
LIN {X 0,Y 298.942,Z 589.734,A -85,B 0,C 180,E1 -16419.403,E2 -16419.403} C_VEL
LIN {X 0,Y 299.406,Z 586.121,A -85,B 0,C 180,E1 -16421.31,E2 -16421.31} C_VEL
LIN {X 0,Y 300.062,Z 580.889,A -85,B 0,C 180,E1 -16423.441,E2 -16423.441} C_VEL
LIN {X 0,Y 300.934,Z 573.442,A -85,B 0,C 180,E1 -16425.811,E2 -16425.811} C_VEL
LIN {X 0,Y 301.957,Z 565.69,A -85,B 0,C 180,E1 -16427.755,E2 -16427.755} C_VEL
LIN {X 0,Y 303.051,Z 556.424,A -85,B 0,C 180,E1 -16429.638,E2 -16429.638} C_VEL
LIN {X 0,Y 304.19,Z 546.374,A -85,B 0,C 180,E1 -16431.299,E2 -16431.299} C_VEL
LIN {X 0,Y 305.206,Z 535.002,A -85,B 0,C 180,E1 -16432.809,E2 -16432.809} C_VEL
LIN {X 0,Y 302.213,Z 523.834,A -85,B 0,C 180,E1 -16434.247,E2 -16434.247} C_VEL
LIN {X 0,Y 298.455,Z 511.311,A -85,B 0,C 180,E1 -16435.587,E2 -16435.587} C_VEL
LIN {X 0,Y 298.4,Z 511.315,A -85,B 0,C 180,E1 -16438.791,E2 -16438.791} C_VEL
LIN {X 0,Y 298.474,Z 511.305,A -85,B 0,C 180,E1 -16441.905,E2 -16441.905} C_VEL
LIN {X 0,Y 298.489,Z 511.303,A -85,B 0,C 180,E1 -16444.924,E2 -16444.924} C_VEL
LIN {X 0,Y 298.434,Z 511.313,A -85,B 0,C 180,E1 -16449.314,E2 -16449.314} C_VEL
LIN {X 0,Y 298.508,Z 511.299,A -85,B 0,C 180,E1 -16452.177,E2 -16452.177} C_VEL
LIN {X 0,Y 298.59,Z 511.291,A -85,B 0,C 180,E1 -16454.994,E2 -16454.994} C_VEL
LIN {X 0,Y 298.589,Z 511.293,A -85,B 0,C 180,E1 -16459.146,E2 -16459.146} C_VEL
LIN {X 0,Y 298.703,Z 511.275,A -85,B 0,C 180,E1 -16461.884,E2 -16461.884} C_VEL
LIN {X 0,Y 298.645,Z 511.282,A -85,B 0,C 180,E1 -16464.598,E2 -16464.598} C_VEL
LIN {X 0,Y 298.922,Z 511.248,A -85,B 0,C 180,E1 -16468.653,E2 -16468.653} C_VEL
LIN {X 0,Y 298.925,Z 511.251,A -85,B 0,C 180,E1 -16471.347,E2 -16471.347} C_VEL
LIN {X 0,Y 298.64,Z 511.286,A -85,B 0,C 180,E1 -16475.401,E2 -16475.401} C_VEL
LIN {X 0,Y 298.712,Z 511.274,A -85,B 0,C 180,E1 -16478.82,E2 -16478.82} C_VEL
LIN {X 0,Y 298.55,Z 511.295,A -85,B 0,C 180,E1 -16483.615,E2 -16483.615} C_VEL
LIN {X 0,Y 298.491,Z 511.3,A -85,B 0,C 180,E1 -16486.412,E2 -16486.412} C_VEL
LIN {X 0,Y 298.503,Z 511.301,A -85,B 0,C 180,E1 -16489.648,E2 -16489.648} C_VEL
LIN {X 0,Y 298.43,Z 511.31,A -85,B 0,C 180,E1 -16493.6,E2 -16493.6} C_VEL
LIN {X 0,Y 298.42,Z 511.31,A -85,B 0,C 180,E1 -16496.581,E2 -16496.581} C_VEL
LIN {X 0,Y 298.403,Z 511.313,A -85,B 0,C 180,E1 -16499.643,E2 -16499.643} C_VEL
LIN {X 0,Y 298.396,Z 511.315,A -85,B 0,C 180,E1 -16502.8,E2 -16502.8} C_VEL
LIN {X 0,Y 298.444,Z 511.309,A -85,B 0,C 180,E1 -16506.806,E2 -16506.806} C_VEL
LIN {X 0,Y 298.351,Z 511.323,A -85,B 0,C 180,E1 -16511.079,E2 -16511.079} C_VEL
LIN {X 0,Y 298.401,Z 511.316,A -85,B 0,C 180,E1 -16513.103,E2 -16513.103} C_VEL
LIN {X 0,Y 298.405,Z 511.315,A -85,B 0,C 180,E1 -16516.92,E2 -16516.92} C_VEL
LIN {X 0,Y 298.401,Z 511.316,A -85,B 0,C 180,E1 -16521.007,E2 -16521.007} C_VEL
LIN {X 0,Y 298.42,Z 511.309,A -85,B 0,C 180,E1 -16523.93,E2 -16523.93} C_VEL
LIN {X 0,Y 298.398,Z 511.312,A -85,B 0,C 180,E1 -16527.983,E2 -16527.983} C_VEL
LIN {X 0,Y 298.466,Z 511.304,A -85,B 0,C 180,E1 -16531.904,E2 -16531.904} C_VEL
LIN {X 0,Y 298.486,Z 511.306,A -85,B 0,C 180,E1 -16534.924,E2 -16534.924} C_VEL
LIN {X 0,Y 298.442,Z 511.309,A -85,B 0,C 180,E1 -16539.314,E2 -16539.314} C_VEL
LIN {X 0,Y 298.54,Z 511.295,A -85,B 0,C 180,E1 -16542.179,E2 -16542.179} C_VEL
LIN {X 0,Y 298.596,Z 511.293,A -85,B 0,C 180,E1 -16544.994,E2 -16544.994} C_VEL
LIN {X 0,Y 298.585,Z 511.293,A -85,B 0,C 180,E1 -16549.146,E2 -16549.146} C_VEL
LIN {X 0,Y 298.704,Z 511.274,A -85,B 0,C 180,E1 -16551.884,E2 -16551.884} C_VEL
LIN {X 0,Y 298.643,Z 511.284,A -85,B 0,C 180,E1 -16554.598,E2 -16554.598} C_VEL
LIN {X 0,Y 298.921,Z 511.25,A -85,B 0,C 180,E1 -16558.652,E2 -16558.652} C_VEL
LIN {X 0,Y 298.92,Z 511.248,A -85,B 0,C 180,E1 -16561.281,E2 -16561.281} C_VEL
LIN {X 0,Y 298.257,Z 511.339,A -85,B 0,C 180,E1 -16562.402,E2 -16562.402} C_VEL
LIN {X 0,Y 295.357,Z 511.706,A -85,B 0,C 180,E1 -16564.226,E2 -16564.226} C_VEL
LIN {X 0,Y 292.868,Z 512.012,A -85,B 0,C 180,E1 -16565.705,E2 -16565.705} C_VEL
LIN {X 0,Y 291.77,Z 512.143,A -85,B 0,C 180,E1 -16566.853,E2 -16566.853} C_VEL
LIN {X 0,Y 291.665,Z 512.153,A -85,B 0,C 180,E1 -16567.243,E2 -16567.243} C_VEL
LIN {X 0,Y 291.574,Z 512.162,A -85,B 0,C 180,E1 -16569.713,E2 -16569.713} C_VEL
LIN {X 0,Y 291.518,Z 512.169,A -85,B 0,C 180,E1 -16573.95,E2 -16573.95} C_VEL
LIN {X 0,Y 291.44,Z 512.18,A -85,B 0,C 180,E1 -16578.269,E2 -16578.269} C_VEL
LIN {X 0,Y 291.36,Z 512.19,A -85,B 0,C 180,E1 -16581.212,E2 -16581.212} C_VEL
LIN {X 0,Y 291.366,Z 512.189,A -85,B 0,C 180,E1 -16584.208,E2 -16584.208} C_VEL
LIN {X 0,Y 291.359,Z 512.19,A -85,B 0,C 180,E1 -16587.278,E2 -16587.278} C_VEL
LIN {X 0,Y 291.321,Z 512.196,A -85,B 0,C 180,E1 -16590.439,E2 -16590.439} C_VEL
LIN {X 0,Y 291.344,Z 512.191,A -85,B 0,C 180,E1 -16593.698,E2 -16593.698} C_VEL
LIN {X 0,Y 291.376,Z 512.189,A -85,B 0,C 180,E1 -16597.254,E2 -16597.254} C_VEL
LIN {X 0,Y 291.413,Z 512.359,A -85,B 0,C 180,E1 -16600.468,E2 -16600.468} C_VEL
LIN {X 0,Y 292.803,Z 519.516,A -85,B 0,C 180,E1 -16604.112,E2 -16604.112} C_VEL
LIN {X 0,Y 294.362,Z 527.678,A -85,B 0,C 180,E1 -16608.048,E2 -16608.048} C_VEL
LIN {X 0,Y 295.579,Z 533.863,A -85,B 0,C 180,E1 -16610.908,E2 -16610.908} C_VEL
LIN {X 0,Y 295.76,Z 535.988,A -85,B 0,C 180,E1 -16611.843,E2 -16611.843} C_VEL
LIN {X 0,Y 294.519,Z 543.639,A -85,B 0,C 180,E1 -16615.061,E2 -16615.061} C_VEL
LIN {X 0,Y 293.459,Z 551.21,A -85,B 0,C 180,E1 -16618.206,E2 -16618.206} C_VEL
LIN {X 0,Y 291.981,Z 562.797,A -85,B 0,C 180,E1 -16622.948,E2 -16622.948} C_VEL
LIN {X 0,Y 291.108,Z 571.792,A -85,B 0,C 180,E1 -16626.572,E2 -16626.572} C_VEL
LIN {X 0,Y 292.582,Z 586.462,A -85,B 0,C 180,E1 -16627.342,E2 -16627.342} C_VEL
LIN {X 0,Y 293.483,Z 599.449,A -85,B 0,C 180,E1 -16628.286,E2 -16628.286} C_VEL
LIN {X 0,Y 294.04,Z 610.912,A -85,B 0,C 180,E1 -16629.357,E2 -16629.357} C_VEL
LIN {X 0,Y 294.287,Z 623.577,A -85,B 0,C 180,E1 -16630.83,E2 -16630.83} C_VEL
LIN {X 0,Y 294.082,Z 632.402,A -85,B 0,C 180,E1 -16632.08,E2 -16632.08} C_VEL
LIN {X 0,Y 292.935,Z 641.155,A -85,B 0,C 180,E1 -16633.539,E2 -16633.539} C_VEL
LIN {X 0,Y 291.736,Z 650.061,A -85,B 0,C 180,E1 -16635.348,E2 -16635.348} C_VEL
LIN {X 0,Y 290.954,Z 658.355,A -85,B 0,C 180,E1 -16637.444,E2 -16637.444} C_VEL
LIN {X 0,Y 290.533,Z 665.036,A -85,B 0,C 180,E1 -16639.547,E2 -16639.547} C_VEL
LIN {X 0,Y 290.471,Z 670.349,A -85,B 0,C 180,E1 -16641.653,E2 -16641.653} C_VEL
LIN {X 0,Y 290.6,Z 674.424,A -85,B 0,C 180,E1 -16643.752,E2 -16643.752} C_VEL
LIN {X 0,Y 290.876,Z 677.373,A -85,B 0,C 180,E1 -16645.843,E2 -16645.843} C_VEL
LIN {X 0,Y 291.013,Z 678.744,A -85,B 0,C 180,E1 -16647.232,E2 -16647.232} C_VEL
LIN {X 0,Y 291.251,Z 679.66,A -85,B 0,C 180,E1 -16648.617,E2 -16648.617} C_VEL
LIN {X 0,Y 291.475,Z 680.146,A -85,B 0,C 180,E1 -16650,E2 -16650} C_VEL
LIN {X 0,Y 291.086,Z 680.118,A -85,B 0,C 180,E1 -16651.384,E2 -16651.384} C_VEL
LIN {X 0,Y 290.911,Z 679.67,A -85,B 0,C 180,E1 -16652.77,E2 -16652.77} C_VEL
LIN {X 0,Y 290.781,Z 678.787,A -85,B 0,C 180,E1 -16654.158,E2 -16654.158} C_VEL
LIN {X 0,Y 290.351,Z 675.747,A -85,B 0,C 180,E1 -16656.952,E2 -16656.952} C_VEL
LIN {X 0,Y 290.217,Z 672.303,A -85,B 0,C 180,E1 -16659.057,E2 -16659.057} C_VEL
LIN {X 0,Y 290.423,Z 667.833,A -85,B 0,C 180,E1 -16661.163,E2 -16661.163} C_VEL
LIN {X 0,Y 291.195,Z 661.204,A -85,B 0,C 180,E1 -16663.611,E2 -16663.611} C_VEL
LIN {X 0,Y 292.016,Z 655.404,A -85,B 0,C 180,E1 -16665.352,E2 -16665.352} C_VEL
LIN {X 0,Y 293.663,Z 647.083,A -85,B 0,C 180,E1 -16667.407,E2 -16667.407} C_VEL
LIN {X 0,Y 295.369,Z 638.782,A -85,B 0,C 180,E1 -16669.097,E2 -16669.097} C_VEL
LIN {X 0,Y 296.275,Z 633.041,A -85,B 0,C 180,E1 -16670.118,E2 -16670.118} C_VEL
LIN {X 0,Y 297.374,Z 621.919,A -85,B 0,C 180,E1 -16671.853,E2 -16671.853} C_VEL
LIN {X 0,Y 298.158,Z 609.969,A -85,B 0,C 180,E1 -16673.39,E2 -16673.39} C_VEL
LIN {X 0,Y 298.021,Z 597.41,A -85,B 0,C 180,E1 -16674.797,E2 -16674.797} C_VEL
LIN {X 0,Y 296.762,Z 584.812,A -85,B 0,C 180,E1 -16676.057,E2 -16676.057} C_VEL
LIN {X 0,Y 294.531,Z 571.751,A -85,B 0,C 180,E1 -16677.22,E2 -16677.22} C_VEL
LIN {X 0,Y 292.661,Z 564.171,A -85,B 0,C 180,E1 -16677.874,E2 -16677.874} C_VEL
LIN {X 0,Y 292.271,Z 561.551,A -85,B 0,C 180,E1 -16678.079,E2 -16678.079} C_VEL
LIN {X 0,Y 293.409,Z 552.636,A -85,B 0,C 180,E1 -16681.801,E2 -16681.801} C_VEL
LIN {X 0,Y 295.036,Z 543.168,A -85,B 0,C 180,E1 -16685.913,E2 -16685.913} C_VEL
LIN {X 0,Y 296.098,Z 537.614,A -85,B 0,C 180,E1 -16688.439,E2 -16688.439} C_VEL
LIN {X 0,Y 295.53,Z 532.576,A -85,B 0,C 180,E1 -16691.042,E2 -16691.042} C_VEL
LIN {X 0,Y 294.499,Z 526.854,A -85,B 0,C 180,E1 -16694.281,E2 -16694.281} C_VEL
LIN {X 0,Y 293.285,Z 521.046,A -85,B 0,C 180,E1 -16697.976,E2 -16697.976} C_VEL
LIN {X 0,Y 292.282,Z 516.436,A -85,B 0,C 180,E1 -16701.305,E2 -16701.305} C_VEL
LIN {X 0,Y 291.379,Z 512.191,A -85,B 0,C 180,E1 -16704.924,E2 -16704.924} C_VEL
LIN {X 0,Y 291.374,Z 512.185,A -85,B 0,C 180,E1 -16707.951,E2 -16707.951} C_VEL
LIN {X 0,Y 291.384,Z 512.182,A -85,B 0,C 180,E1 -16711.159,E2 -16711.159} C_VEL
LIN {X 0,Y 291.42,Z 512.181,A -85,B 0,C 180,E1 -16714.272,E2 -16714.272} C_VEL
LIN {X 0,Y 291.384,Z 512.187,A -85,B 0,C 180,E1 -16717.3,E2 -16717.3} C_VEL
LIN {X 0,Y 291.46,Z 512.179,A -85,B 0,C 180,E1 -16720.271,E2 -16720.271} C_VEL
LIN {X 0,Y 291.558,Z 512.163,A -85,B 0,C 180,E1 -16724.624,E2 -16724.624} C_VEL
LIN {X 0,Y 291.54,Z 512.163,A -85,B 0,C 180,E1 -16728.881,E2 -16728.881} C_VEL
LIN {X 0,Y 291.713,Z 512.141,A -85,B 0,C 180,E1 -16731.689,E2 -16731.689} C_VEL
LIN {X 0,Y 291.629,Z 512.154,A -85,B 0,C 180,E1 -16734.469,E2 -16734.469} C_VEL
LIN {X 0,Y 291.888,Z 512.126,A -85,B 0,C 180,E1 -16738.621,E2 -16738.621} C_VEL
LIN {X 0,Y 291.892,Z 512.127,A -85,B 0,C 180,E1 -16741.38,E2 -16741.38} C_VEL
LIN {X 0,Y 291.713,Z 512.337,A -85,B 0,C 180,E1 -16746.702,E2 -16746.702} C_VEL
LIN {X 0,Y 292.212,Z 514.017,A -85,B 0,C 180,E1 -16746.907,E2 -16746.907} C_VEL
LIN {X 0,Y 296.653,Z 522.651,A -85,B 0,C 180,E1 -16748.358,E2 -16748.358} C_VEL
LIN {X 0,Y 300.809,Z 532.904,A -85,B 0,C 180,E1 -16750.092,E2 -16750.092} C_VEL
LIN {X 0,Y 303.655,Z 541.951,A -85,B 0,C 180,E1 -16751.696,E2 -16751.696} C_VEL
LIN {X 0,Y 304.781,Z 547.184,A -85,B 0,C 180,E1 -16752.654,E2 -16752.654} C_VEL
LIN {X 0,Y 302.961,Z 557.18,A -85,B 0,C 180,E1 -16754.218,E2 -16754.218} C_VEL
LIN {X 0,Y 301.096,Z 565.94,A -85,B 0,C 180,E1 -16755.918,E2 -16755.918} C_VEL
LIN {X 0,Y 298.962,Z 575.044,A -85,B 0,C 180,E1 -16758.149,E2 -16758.149} C_VEL
LIN {X 0,Y 297.438,Z 581.125,A -85,B 0,C 180,E1 -16760.036,E2 -16760.036} C_VEL
LIN {X 0,Y 295.769,Z 586.939,A -85,B 0,C 180,E1 -16762.346,E2 -16762.346} C_VEL
LIN {X 0,Y 294.308,Z 591.564,A -85,B 0,C 180,E1 -16764.846,E2 -16764.846} C_VEL
LIN {X 0,Y 293.163,Z 594.781,A -85,B 0,C 180,E1 -16767.5,E2 -16767.5} C_VEL
LIN {X 0,Y 292.299,Z 596.524,A -85,B 0,C 180,E1 -16770.327,E2 -16770.327} C_VEL
LIN {X 0,Y 291.875,Z 596.717,A -85,B 0,C 180,E1 -16772.567,E2 -16772.567} C_VEL
LIN {X 0,Y 291.664,Z 595.49,A -85,B 0,C 180,E1 -16775.332,E2 -16775.332} C_VEL
LIN {X 0,Y 291.688,Z 593.623,A -85,B 0,C 180,E1 -16777.334,E2 -16777.334} C_VEL
LIN {X 0,Y 291.937,Z 590.412,A -85,B 0,C 180,E1 -16779.613,E2 -16779.613} C_VEL
LIN {X 0,Y 292.498,Z 586.044,A -85,B 0,C 180,E1 -16781.853,E2 -16781.853} C_VEL
LIN {X 0,Y 293.206,Z 580.509,A -85,B 0,C 180,E1 -16784.037,E2 -16784.037} C_VEL
LIN {X 0,Y 294.16,Z 572.796,A -85,B 0,C 180,E1 -16786.411,E2 -16786.411} C_VEL
LIN {X 0,Y 295.258,Z 564.604,A -85,B 0,C 180,E1 -16788.414,E2 -16788.414} C_VEL
LIN {X 0,Y 296.365,Z 555.732,A -85,B 0,C 180,E1 -16790.187,E2 -16790.187} C_VEL
LIN {X 0,Y 297.546,Z 545.139,A -85,B 0,C 180,E1 -16791.898,E2 -16791.898} C_VEL
LIN {X 0,Y 298.324,Z 536.967,A -85,B 0,C 180,E1 -16792.998,E2 -16792.998} C_VEL
LIN {X 0,Y 295.687,Z 526.539,A -85,B 0,C 180,E1 -16794.385,E2 -16794.385} C_VEL
LIN {X 0,Y 292.015,Z 514.342,A -85,B 0,C 180,E1 -16795.766,E2 -16795.766} C_VEL
LIN {X 0,Y 291.398,Z 512.188,A -85,B 0,C 180,E1 -16795.996,E2 -16795.996} C_VEL
LIN {X 0,Y 291.392,Z 512.187,A -85,B 0,C 180,E1 -16800.26,E2 -16800.26} C_VEL
LIN {X 0,Y 291.424,Z 512.182,A -85,B 0,C 180,E1 -16804.272,E2 -16804.272} C_VEL
LIN {X 0,Y 291.377,Z 512.192,A -85,B 0,C 180,E1 -16807.299,E2 -16807.299} C_VEL
LIN {X 0,Y 291.444,Z 512.179,A -85,B 0,C 180,E1 -16810.269,E2 -16810.269} C_VEL
LIN {X 0,Y 291.502,Z 512.172,A -85,B 0,C 180,E1 -16814.665,E2 -16814.665} C_VEL
LIN {X 0,Y 291.534,Z 512.169,A -85,B 0,C 180,E1 -16818.88,E2 -16818.88} C_VEL
LIN {X 0,Y 291.656,Z 512.154,A -85,B 0,C 180,E1 -16821.687,E2 -16821.687} C_VEL
LIN {X 0,Y 291.613,Z 512.158,A -85,B 0,C 180,E1 -16824.468,E2 -16824.468} C_VEL
LIN {X 0,Y 291.889,Z 512.124,A -85,B 0,C 180,E1 -16828.62,E2 -16828.62} C_VEL
LIN {X 0,Y 291.891,Z 512.127,A -85,B 0,C 180,E1 -16831.379,E2 -16831.379} C_VEL
LIN {X 0,Y 291.609,Z 512.161,A -85,B 0,C 180,E1 -16835.532,E2 -16835.532} C_VEL
LIN {X 0,Y 291.671,Z 512.152,A -85,B 0,C 180,E1 -16838.91,E2 -16838.91} C_VEL
LIN {X 0,Y 291.521,Z 512.169,A -85,B 0,C 180,E1 -16842.531,E2 -16842.531} C_VEL
LIN {X 0,Y 291.511,Z 512.173,A -85,B 0,C 180,E1 -16845.379,E2 -16845.379} C_VEL
LIN {X 0,Y 291.455,Z 512.178,A -85,B 0,C 180,E1 -16849.874,E2 -16849.874} C_VEL
LIN {X 0,Y 291.372,Z 512.187,A -85,B 0,C 180,E1 -16854.208,E2 -16854.208} C_VEL
LIN {X 0,Y 291.366,Z 512.193,A -85,B 0,C 180,E1 -16857.277,E2 -16857.277} C_VEL
LIN {X 0,Y 291.326,Z 512.194,A -85,B 0,C 180,E1 -16860.438,E2 -16860.438} C_VEL
LIN {X 0,Y 291.347,Z 512.191,A -85,B 0,C 180,E1 -16863.698,E2 -16863.698} C_VEL
LIN {X 0,Y 291.372,Z 512.192,A -85,B 0,C 180,E1 -16867.252,E2 -16867.252} C_VEL
LIN {X 0,Y 291.303,Z 512.198,A -85,B 0,C 180,E1 -16870.648,E2 -16870.648} C_VEL
LIN {X 0,Y 291.292,Z 512.197,A -85,B 0,C 180,E1 -16874.402,E2 -16874.402} C_VEL
LIN {X 0,Y 291.329,Z 512.193,A -85,B 0,C 180,E1 -16878.404,E2 -16878.404} C_VEL
LIN {X 0,Y 291.35,Z 512.194,A -85,B 0,C 180,E1 -16881.157,E2 -16881.157} C_VEL
LIN {X 0,Y 291.363,Z 512.19,A -85,B 0,C 180,E1 -16884.626,E2 -16884.626} C_VEL
LIN {X 0,Y 291.375,Z 512.187,A -85,B 0,C 180,E1 -16887.95,E2 -16887.95} C_VEL
LIN {X 0,Y 291.385,Z 512.19,A -85,B 0,C 180,E1 -16891.158,E2 -16891.158} C_VEL
LIN {X 0,Y 291.418,Z 512.182,A -85,B 0,C 180,E1 -16894.271,E2 -16894.271} C_VEL
LIN {X 0,Y 291.376,Z 512.189,A -85,B 0,C 180,E1 -16897.299,E2 -16897.299} C_VEL
LIN {X 0,Y 291.46,Z 512.176,A -85,B 0,C 180,E1 -16900.27,E2 -16900.27} C_VEL
LIN {X 0,Y 291.557,Z 512.167,A -85,B 0,C 180,E1 -16904.623,E2 -16904.623} C_VEL
LIN {X 0,Y 291.531,Z 512.172,A -85,B 0,C 180,E1 -16908.88,E2 -16908.88} C_VEL
LIN {X 0,Y 291.657,Z 512.152,A -85,B 0,C 180,E1 -16911.687,E2 -16911.687} C_VEL
LIN {X 0,Y 291.611,Z 512.159,A -85,B 0,C 180,E1 -16914.468,E2 -16914.468} C_VEL
LIN {X 0,Y 291.887,Z 512.126,A -85,B 0,C 180,E1 -16918.62,E2 -16918.62} C_VEL
LIN {X 0,Y 291.887,Z 512.125,A -85,B 0,C 180,E1 -16921.379,E2 -16921.379} C_VEL
LIN {X 0,Y 291.689,Z 512.153,A -85,B 0,C 180,E1 -16926.919,E2 -16926.919} C_VEL
LIN {X 0,Y 291.665,Z 512.153,A -85,B 0,C 180,E1 -16927.243,E2 -16927.243} C_VEL
LIN {X 0,Y 290.948,Z 512.244,A -85,B 0,C 180,E1 -16928.395,E2 -16928.395} C_VEL
LIN {X 0,Y 288.044,Z 512.603,A -85,B 0,C 180,E1 -16930.269,E2 -16930.269} C_VEL
LIN {X 0,Y 285.598,Z 512.91,A -85,B 0,C 180,E1 -16931.79,E2 -16931.79} C_VEL
LIN {X 0,Y 284.542,Z 513.042,A -85,B 0,C 180,E1 -16932.97,E2 -16932.97} C_VEL
LIN {X 0,Y 284.452,Z 513.049,A -85,B 0,C 180,E1 -16933.37,E2 -16933.37} C_VEL
LIN {X 0,Y 284.388,Z 513.059,A -85,B 0,C 180,E1 -16937.25,E2 -16937.25} C_VEL
LIN {X 0,Y 284.368,Z 513.06,A -85,B 0,C 180,E1 -16940.243,E2 -16940.243} C_VEL
LIN {X 0,Y 284.325,Z 513.065,A -85,B 0,C 180,E1 -16943.855,E2 -16943.855} C_VEL
LIN {X 0,Y 284.289,Z 513.07,A -85,B 0,C 180,E1 -16948.015,E2 -16948.015} C_VEL
LIN {X 0,Y 284.286,Z 513.073,A -85,B 0,C 180,E1 -16951.275,E2 -16951.275} C_VEL
LIN {X 0,Y 284.341,Z 513.065,A -85,B 0,C 180,E1 -16955.348,E2 -16955.348} C_VEL
LIN {X 0,Y 284.313,Z 513.069,A -85,B 0,C 180,E1 -16958.169,E2 -16958.169} C_VEL
LIN {X 0,Y 284.385,Z 513.26,A -85,B 0,C 180,E1 -16960.097,E2 -16960.097} C_VEL
LIN {X 0,Y 285.651,Z 519.844,A -85,B 0,C 180,E1 -16963.543,E2 -16963.543} C_VEL
LIN {X 0,Y 287.096,Z 527.292,A -85,B 0,C 180,E1 -16967.255,E2 -16967.255} C_VEL
LIN {X 0,Y 288.639,Z 535.6,A -85,B 0,C 180,E1 -16971.184,E2 -16971.184} C_VEL
LIN {X 0,Y 288.506,Z 538.529,A -85,B 0,C 180,E1 -16972.483,E2 -16972.483} C_VEL
LIN {X 0,Y 286.664,Z 549.922,A -85,B 0,C 180,E1 -16977.36,E2 -16977.36} C_VEL
LIN {X 0,Y 285.105,Z 561.085,A -85,B 0,C 180,E1 -16982.072,E2 -16982.072} C_VEL
